# B&R Automation Studio project mVTest1
Automation Studio 4.12.6.106; technology packages: mappCockpit 5.24.2, mappMotion 5.29.0, mappView 5.24.6

## Configuration Config1

CPU X20CP3687X, AutomationRuntime J4.93, Build 4.1.2, Safety 0.0, Vc V4.73.2

### Task classes (Cpu.sw)
```
Cyclic#1:
  motionprg1 <- motionprg1.prg
  motionprg2 <- motionprg2.prg
Cyclic#4:
  Program <- Program.prg
DataObjects: McAcpSys
NcDataObjects: McDriveLog
Binaries: arsvcreg, udbdef, mvLoader, arflatprv, McAcpDrv, arcoal, FWRules, TCData, mCoWebSc, McAcpSim, Settings, Config_1, ashwac, User, sysconf, asfw, arconfig, Config_3, ashwd, Config_2, iomap, Role
Libraries: arssl, astime, asieccon, mpaxis, powerlnk, runtime, mcaxis, fileio, mpbase, mcbase, sys_lib, CoTrace, AsZip
```

### Hardware
```
X20CP3687X : X20CP3687X v1.6.2.0
  Connector IF2:
    ActivateDevice = 1
    Mode = Manual
    InternetAddress = 192.168.1.50
    SubnetMask = 255.255.255.0
  ConfigurationID = mVTest1_Config1
  FileDevice1
  FileDeviceName1 = USER
  FileDevicePath1 = USER_PATH
  ActivateOpcUa = 1
  OpcUa_AuthenticationSecurityPolicy_EnableNone = 1
  OpcUa_AuthenticationSecurityPolicy_EnableBasic128Rsa15 = 1
  OpcUaInformationModels_PV_Version = 1
```

### Config_2.axis - X20CP3687X/mappMotion/Config_2.axis
```
Element gAxis_2 (Type=axis)
  BaseTypeIsReadOnly = 0
  BaseType = Rotary
    MeasurementUnitIsReadOnly = 0
    MeasurementUnit = 17476
    MeasurementResolutionIsReadOnly = 0
    MeasurementResolution = 0.01
    CountDirectionIsReadOnly = 0
    CountDirection = Standard
  MovementLimitsIsReadOnly = 0
  MovementLimits = Internal
    Position:
      LowerLimitMin = -1.79769313486231E308
      UpperLimitMax = 1.79769313486231E308
      LowerLimit = -1000.0
      UpperLimit = 1000.0
    VelocityIsReadOnly = 0
    Velocity:
      VelocityMax = 3.4E38
      Velocity = 30
    AccelerationIsReadOnly = 0
    Acceleration:
      AccelerationMax = 3.4E38
      Acceleration = 50.0
    DecelerationIsReadOnly = 0
    Deceleration:
      DecelerationMax = 3.4E38
      Deceleration = 50.0
  Alarms = None
```

## Configuration Config2

CPU PC_any, AutomationRuntime J4.93, Build 4.1.2, Vc V4.73.2

### Hardware
```
PC : PC_any v1.1.1.0 (OrderNumber=PC)
  ConfigurationID = mVTest1_Config2
  FileDevice1
  FileDeviceName1 = USER
  FileDevicePath1 = USER_PATH
  ActivateOpcUa = 1
  OpcUaInformationModels_PV_Version = 1
```

## Configuration Config3

CPU 4PPC50.101E-10B, AutomationRuntime J4.93, Build 4.1.2, Safety 0.0, Vc V4.73.2

### Task classes (Cpu.sw)
```
Cyclic#1 (cycle 2000 us, tolerance 2000 us):
  motionprg1 <- motionprg1.prg
  motionprg2 <- motionprg2.prg
Cyclic#2 (cycle 20000 us, tolerance 20000 us):
  room3 <- room.prg
  room1 <- room.prg
  room2 <- room.prg
Cyclic#4 (cycle 100000 us, tolerance 100000 us):
  Program <- Program.prg
  tcp <- tcp.prg
DataObjects: McAcpSys
NcDataObjects: McDriveLog
Binaries: arsvcreg, udbdef, mvLoader, arflatprv, McAcpDrv, arcoal, FWRules, TCData, mCoWebSc, McAcpSim, Settings, Config_1, ashwac, User, sysconf, asfw, arconfig, iomap, Config_3, ashwd, Config_2, Role
Libraries: McBase, MpBase, MpAxis, McAxis, McAcpAx, CoTrace, AsZip, FileIO, runtime, AsTCP, helper, arssl, astime, asieccon, powerlnk, asepl, sys_lib
```

### Hardware
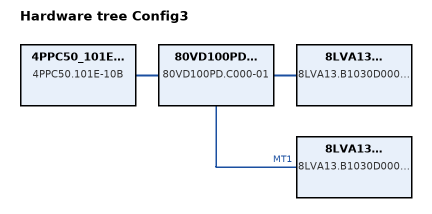
```
4PPC50_101E_10B : 4PPC50.101E-10B v1.1.4.0
  Connector IF2:
    ActivateDevice = 1
    Mode = Manual
    InternetAddress = 192.168.1.50
    SubnetMask = 255.255.255.0
    ActivateSnmp = 1
  Connector IF3:
    AssignedOperatingSystem = ARemb
  Connector IF4:
    AssignedOperatingSystem = GPOS
  ConfigurationID = mVTest1_Config3
  TimerDeviceType = EPLX2X
  TimerDevice = 4PPC50_101E_10B.IF1
  TaskClassIdleTime = 2000
  Cyclic1Duration = 2000
  Cyclic1Tolerance = 2000
  Cyclic2Duration = 20000
  Cyclic2Tolerance = 20000
  Cyclic3Duration = 50000
  Cyclic3Tolerance = 50000
  Cyclic4Duration = 100000
  Cyclic4Tolerance = 100000
  Cyclic5Duration = 200000
  Cyclic5Tolerance = 200000
  Cyclic6Duration = 500000
  Cyclic6Tolerance = 500000
  Cyclic7Duration = 1000000
  Cyclic7Tolerance = 1000000
  Cyclic8Duration = 10000
  Cyclic8Tolerance = 30000000
  FileDevice1
  FileDeviceName1 = USER
  FileDevicePath1 = USER_PATH
  ActivateOpcUa = 1
  OpcUa_AuthenticationSecurityPolicy_EnableNone = 1
  OpcUa_AuthenticationSecurityPolicy_EnableBasic128Rsa15 = 1
  OpcUaInformationModels_PV_Version = 1
  LXTMode = Manual
  LXTInternetAddress = 192.168.1.51
  LXTSubnetmask = 255.255.255.0
  LXTVisuURL = 192.168.1.50:81/index.html
80VD100PD.C000-01 : 80VD100PD.C000-01 v2.5.0.0  [PLK1 -> 4PPC50_101E_10B.IF1 (NodeNumber=1) [Cable Type=PowerlinkCable, Length=10, Version=1.0.0.3]; MT2 -> 8LVA13.B1030D000-0.MT]
  DriveConfiguration/Module:
    McAcoposTypeID = AcoposMicroDConfig
    ActivateACOPOSSimulationOnPLC = 0
  DriveConfiguration/Channel[1]/RealAxis:
    AxisReference = gAxis_1
    MechanicalElementsIsInvisible = 0
  DriveConfiguration/Channel[1]/RealAxis/MechanicalElements/Gearbox:
    InputIsReadOnly = 0
    Input = 1
    OutputIsReadOnly = 0
    Output = 1
  DriveConfiguration/Channel[1]/RealAxis/MechanicalElements/RotaryToLinearTransformation:
    ReferenceDistanceIsReadOnly = 0
    ReferenceDistance = 1
  DriveConfiguration/Channel[1]/RealAxis/Controller:
    ModeIsReadOnly = 0
    Mode = PositionController
  DriveConfiguration/Channel[1]/RealAxis/Controller/Mode/Position:
    ProportionalGain = 50.0
    IntegrationTime = 0.0
    PredictionTime = 0.0004
    TotalDelayTime = 0.0004
  DriveConfiguration/Channel[1]/RealAxis/Controller/Mode/Speed:
    ProportionalGainIsReadOnly = 0
    ProportionalGain = 2.0
    IntegrationTimeIsReadOnly = 0
    IntegrationTime = 0.0
    FilterTimeIsReadOnly = 0
    FilterTime = 0.0
  DriveConfiguration/Channel[1]/RealAxis/Controller/Mode/LoopFilters:
    LoopFilterXIsReadOnly = 0
    LoopFilter1 = NotUsed
    LoopFilter2 = NotUsed
    LoopFilter3 = NotUsed
  DriveConfiguration/Channel[1]/RealAxis/Homing:
    ModeIsReadOnly = 0
    Mode = Direct
  DriveConfiguration/Channel[1]/RealAxis/Homing/Mode:
    Position = 0.0
    ReferencePulse = NotUsed
  DriveConfiguration/Channel[1]/RealAxis/Homing:
    RestorePositionVariable = 
  DriveConfiguration/Channel[1]/RealAxis/StopReaction:
    QuickstopIsReadOnly = 0
    Quickstop = DecelerationLimit
    DriveErrorIsReadOnly = 0
    DriveError = DecelerationLimit
    FilterTime = 10
  DriveConfiguration/Channel[1]/RealAxis/MovementErrorLimits:
    PositionError = 10
    VelocityErrorMonitoring = Automatic1
  DriveConfiguration/Channel[1]/RealAxis:
    JerkFilterIsReadOnly = 0
    JerkFilter = NotUsed
    ZeroVibrationFilter = NotUsed
  DriveConfiguration/Channel[1]/RealAxis/DigitalInputs/HomingSwitch:
    SourceIsReadOnly = 0
    Source = NotUsed
    Level = High
  DriveConfiguration/Channel[1]/RealAxis/DigitalInputs/PositiveLimitSwitch:
    SourceIsReadOnly = 0
    Source = NotUsed
    Level = High
  DriveConfiguration/Channel[1]/RealAxis/DigitalInputs/NegativeLimitSwitch:
    SourceIsReadOnly = 0
    Source = NotUsed
    Level = High
  DriveConfiguration/Channel[1]/RealAxis/DigitalInputs/Trigger1:
    Source = Force
    Level = High
  DriveConfiguration/Channel[1]/RealAxis/DigitalInputs/Trigger2:
    Source = Force
    Level = High
  DriveConfiguration/Channel[1]/RealAxis/DigitalInputs/Quickstop:
    Input = NotUsed
  DriveConfiguration/Channel[1]/RealAxis/Simulation:
    SimulationModeOnPLC = SetValueGeneration
    SimulationModeOnACOPOS = NotUsed
  DriveConfiguration/Channel[1]:
    ExternalEncoderAxis = NotUsed
  DriveConfiguration/Channel[2]/RealAxis:
    AxisReference = gAxis_2
    MechanicalElementsIsInvisible = 0
  DriveConfiguration/Channel[2]/RealAxis/MechanicalElements/Gearbox:
    InputIsReadOnly = 0
    Input = 1
    OutputIsReadOnly = 0
    Output = 1
  DriveConfiguration/Channel[2]/RealAxis/MechanicalElements/RotaryToLinearTransformation:
    ReferenceDistanceIsReadOnly = 0
    ReferenceDistance = 1
  DriveConfiguration/Channel[2]/RealAxis/Controller:
    ModeIsReadOnly = 0
    Mode = PositionController
  DriveConfiguration/Channel[2]/RealAxis/Controller/Mode/Position:
    ProportionalGain = 50.0
    IntegrationTime = 0.0
    PredictionTime = 0.0004
    TotalDelayTime = 0.0004
  DriveConfiguration/Channel[2]/RealAxis/Controller/Mode/Speed:
    ProportionalGainIsReadOnly = 0
    ProportionalGain = 2.0
    IntegrationTimeIsReadOnly = 0
    IntegrationTime = 0.0
    FilterTimeIsReadOnly = 0
    FilterTime = 0.0
  DriveConfiguration/Channel[2]/RealAxis/Controller/Mode/LoopFilters:
    LoopFilterXIsReadOnly = 0
    LoopFilter1 = NotUsed
    LoopFilter2 = NotUsed
    LoopFilter3 = NotUsed
  DriveConfiguration/Channel[2]/RealAxis/Homing:
    ModeIsReadOnly = 0
    Mode = Direct
  DriveConfiguration/Channel[2]/RealAxis/Homing/Mode:
    Position = 0.0
    ReferencePulse = NotUsed
  DriveConfiguration/Channel[2]/RealAxis/Homing:
    RestorePositionVariable = 
  DriveConfiguration/Channel[2]/RealAxis/StopReaction:
    QuickstopIsReadOnly = 0
    Quickstop = DecelerationLimit
    DriveErrorIsReadOnly = 0
    DriveError = DecelerationLimit
    FilterTime = 0.0
  DriveConfiguration/Channel[2]/RealAxis/MovementErrorLimits:
    PositionError = 10
    VelocityErrorMonitoring = Automatic1
  DriveConfiguration/Channel[2]/RealAxis:
    JerkFilterIsReadOnly = 0
    JerkFilter = NotUsed
    ZeroVibrationFilter = NotUsed
  DriveConfiguration/Channel[2]/RealAxis/DigitalInputs/HomingSwitch:
    SourceIsReadOnly = 0
    Source = NotUsed
    Level = High
  DriveConfiguration/Channel[2]/RealAxis/DigitalInputs/PositiveLimitSwitch:
    SourceIsReadOnly = 0
    Source = NotUsed
    Level = High
  DriveConfiguration/Channel[2]/RealAxis/DigitalInputs/NegativeLimitSwitch:
    SourceIsReadOnly = 0
    Source = NotUsed
    Level = High
  DriveConfiguration/Channel[2]/RealAxis/DigitalInputs/Trigger1:
    Source = X2Trigger1
    Level = High
  DriveConfiguration/Channel[2]/RealAxis/DigitalInputs/Trigger2:
    Source = X2Trigger2
    Level = High
  DriveConfiguration/Channel[2]/RealAxis/DigitalInputs/Quickstop:
    Input = NotUsed
  DriveConfiguration/Channel[2]/RealAxis/Simulation:
    SimulationModeOnPLC = SetValueGeneration
    SimulationModeOnACOPOS = NotUsed
  DriveConfiguration/Channel[2]:
    ExternalEncoderAxis = NotUsed
8LVA13.B1030D000-0 : 8LVA13.B1030D000-0 v2.2.0.3  [MT -> 80VD100PD.C000-01.MT2]
  M1/MotorParameters:
    MOTOR_AMB_TEMP_RATED = 40
8LVA13.B1030D000-0a : 8LVA13.B1030D000-0 v2.2.0.3  [MT -> 80VD100PD.C000-01.MT1]
  M1/MotorParameters:
    MOTOR_AMB_TEMP_RATED = 40
```

### Config_1.axis - 4PPC50_101E_10B/mappMotion/Config_1.axis
```
Element gAxis_1 (Type=axis)
  BaseTypeIsReadOnly = 0
  BaseType = Rotary
    MeasurementUnitIsReadOnly = 0
    MeasurementUnit = 17476
    MeasurementResolutionIsReadOnly = 0
    MeasurementResolution = 0.01
    CountDirectionIsReadOnly = 0
    CountDirection = Standard
  MovementLimitsIsReadOnly = 0
  MovementLimits = Internal
    Position:
      LowerLimitMin = -1.79769313486231E308
      UpperLimitMax = 1.79769313486231E308
      LowerLimit = -1000.0
      UpperLimit = 1000.0
    VelocityIsReadOnly = 0
    Velocity:
      VelocityMax = 3.4E38
      Velocity = 10.0
    AccelerationIsReadOnly = 0
    Acceleration:
      AccelerationMax = 3.4E38
      Acceleration = 50.0
    DecelerationIsReadOnly = 0
    Deceleration:
      DecelerationMax = 3.4E38
      Deceleration = 50.0
  Alarms = None
```

### Config_2.axis - 4PPC50_101E_10B/mappMotion/Config_2.axis
```
Element gAxis_2 (Type=axis)
  BaseTypeIsReadOnly = 0
  BaseType = Rotary
    MeasurementUnitIsReadOnly = 0
    MeasurementUnit = 17476
    MeasurementResolutionIsReadOnly = 0
    MeasurementResolution = 0.01
    CountDirectionIsReadOnly = 0
    CountDirection = Standard
  MovementLimitsIsReadOnly = 0
  MovementLimits = Internal
    Position:
      LowerLimitMin = -1.79769313486231E308
      UpperLimitMax = 1.79769313486231E308
      LowerLimit = -1000.0
      UpperLimit = 1000.0
    VelocityIsReadOnly = 0
    Velocity:
      VelocityMax = 3.4E38
      Velocity = 10.0
    AccelerationIsReadOnly = 0
    Acceleration:
      AccelerationMax = 3.4E38
      Acceleration = 50.0
    DecelerationIsReadOnly = 0
    Deceleration:
      DecelerationMax = 3.4E38
      Deceleration = 50.0
  Alarms = None
```

## Configuration Config4

CPU 4PPC80.101E-11A, AutomationRuntime J4.93, Build 4.1.2, Safety 0.0, Vc V4.73.2

### Task classes (Cpu.sw)
```
Cyclic#1 (cycle 2000 us, tolerance 2000 us):
  motionprg1 <- motionprg1.prg
  motionprg2 <- motionprg2.prg
Cyclic#2:
  opctest <- opctest.prg
  room1 <- room.prg
  room3 <- room.prg
  room2 <- room.prg
Cyclic#4:
  Program <- Program.prg
  tcp <- tcp.prg
DataObjects: McAcpSys
NcDataObjects: McDriveLog
Binaries: arsvcreg, udbdef, mvLoader, arflatprv, McAcpDrv, arcoal, FWRules, TCData, mCoWebSc, McAcpSim, Settings, Config_1, ashwac, User, sysconf, asfw, arconfig, iomap, Config_3, ashwd, Config_2, Role
Libraries: McBase, MpBase, MpAxis, McAxis, McAcpAx, CoTrace, AsZip, FileIO, runtime, McAcpPar, sys_lib, brsystem, helper, arssl, astime, asieccon, powerlnk, asepl
```

### Hardware
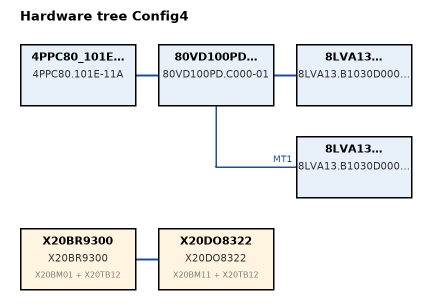
```
4PPC80_101E_11A : 4PPC80.101E-11A v1.0.3.0
  Connector IF2:
    AssignedOperatingSystem = ARemb
    ActivateDevice = 1
    Mode = Manual
    InternetAddress = 192.168.1.51
    SubnetMask = 255.255.255.0
    ActivateSnmp = 1
  Connector IF3:
    OperatingSystem = ARemb
    ActivateDevice = 1
  Connector IF4:
    AssignedOperatingSystem = GPOS
  Connector IF5:
    AssignedOperatingSystem = GPOS
  Connector IF6:
    CycleTime = 4000
  ConfigurationID = mVTest1_Config3
  TimerDeviceType = EPLX2X
  TimerDevice = 4PPC80_101E_11A.IF1
  TaskClassIdleTime = 2000
  Cyclic1Duration = 2000
  Cyclic1Tolerance = 2000
  FileDevice1
  FileDeviceName1 = USER
  FileDevicePath1 = USER_PATH
  ActivateOpcUa = 1
  OpcUa_AuthenticationSecurityPolicy_EnableNone = 1
  OpcUa_AuthenticationSecurityPolicy_EnableBasic128Rsa15 = 1
  OpcUaInformationModels_PV_Version = 1
  LXTVisuURL = 192.168.1.51:81/index.html
80VD100PD.C000-01 : 80VD100PD.C000-01 v2.5.0.0  [PLK1 -> 4PPC80_101E_11A.IF1 (NodeNumber=2) [Cable Type=PowerlinkCable, Length=10, Version=1.0.0.3]; MT2 -> 8LVA13.B1030D000-0.MT]
  DriveConfiguration/Module:
    McAcoposTypeID = AcoposMicroDConfig
    ActivateACOPOSSimulationOnPLC = 0
  DriveConfiguration/Channel[1]/RealAxis:
    AxisReference = gAxis_1
    MechanicalElementsIsInvisible = 0
  DriveConfiguration/Channel[1]/RealAxis/MechanicalElements/Gearbox:
    InputIsReadOnly = 0
    Input = 1
    OutputIsReadOnly = 0
    Output = 1
  DriveConfiguration/Channel[1]/RealAxis/MechanicalElements/RotaryToLinearTransformation:
    ReferenceDistanceIsReadOnly = 0
    ReferenceDistance = 1
  DriveConfiguration/Channel[1]/RealAxis/Controller:
    ModeIsReadOnly = 0
    Mode = PositionController
  DriveConfiguration/Channel[1]/RealAxis/Controller/Mode/Position:
    ProportionalGain = 50.0
    IntegrationTime = 0.0
    PredictionTime = 0.0004
    TotalDelayTime = 0.0004
  DriveConfiguration/Channel[1]/RealAxis/Controller/Mode/Speed:
    ProportionalGainIsReadOnly = 0
    ProportionalGain = 2.0
    IntegrationTimeIsReadOnly = 0
    IntegrationTime = 0.0
    FilterTimeIsReadOnly = 0
    FilterTime = 0.0
  DriveConfiguration/Channel[1]/RealAxis/Controller/Mode/LoopFilters:
    LoopFilterXIsReadOnly = 0
    LoopFilter1 = NotUsed
    LoopFilter2 = NotUsed
    LoopFilter3 = NotUsed
  DriveConfiguration/Channel[1]/RealAxis/Homing:
    ModeIsReadOnly = 0
    Mode = Direct
  DriveConfiguration/Channel[1]/RealAxis/Homing/Mode:
    Position = 0.0
    ReferencePulse = NotUsed
  DriveConfiguration/Channel[1]/RealAxis/Homing:
    RestorePositionVariable = 
  DriveConfiguration/Channel[1]/RealAxis/StopReaction:
    QuickstopIsReadOnly = 0
    Quickstop = DecelerationLimit
    DriveErrorIsReadOnly = 0
    DriveError = DecelerationLimit
    FilterTime = 10
  DriveConfiguration/Channel[1]/RealAxis/MovementErrorLimits:
    PositionError = 10
    VelocityErrorMonitoring = Automatic1
  DriveConfiguration/Channel[1]/RealAxis:
    JerkFilterIsReadOnly = 0
    JerkFilter = NotUsed
    ZeroVibrationFilter = NotUsed
  DriveConfiguration/Channel[1]/RealAxis/DigitalInputs/HomingSwitch:
    SourceIsReadOnly = 0
    Source = NotUsed
    Level = High
  DriveConfiguration/Channel[1]/RealAxis/DigitalInputs/PositiveLimitSwitch:
    SourceIsReadOnly = 0
    Source = NotUsed
    Level = High
  DriveConfiguration/Channel[1]/RealAxis/DigitalInputs/NegativeLimitSwitch:
    SourceIsReadOnly = 0
    Source = NotUsed
    Level = High
  DriveConfiguration/Channel[1]/RealAxis/DigitalInputs/Trigger1:
    Source = Force
    Level = High
  DriveConfiguration/Channel[1]/RealAxis/DigitalInputs/Trigger2:
    Source = Force
    Level = High
  DriveConfiguration/Channel[1]/RealAxis/DigitalInputs/Quickstop:
    Input = NotUsed
  DriveConfiguration/Channel[1]/RealAxis/Simulation:
    SimulationModeOnPLC = SetValueGeneration
    SimulationModeOnACOPOS = NotUsed
  DriveConfiguration/Channel[1]:
    ExternalEncoderAxis = NotUsed
  DriveConfiguration/Channel[2]/RealAxis:
    AxisReference = gAxis_2
    MechanicalElementsIsInvisible = 0
  DriveConfiguration/Channel[2]/RealAxis/MechanicalElements/Gearbox:
    InputIsReadOnly = 0
    Input = 1
    OutputIsReadOnly = 0
    Output = 1
  DriveConfiguration/Channel[2]/RealAxis/MechanicalElements/RotaryToLinearTransformation:
    ReferenceDistanceIsReadOnly = 0
    ReferenceDistance = 1
  DriveConfiguration/Channel[2]/RealAxis/Controller:
    ModeIsReadOnly = 0
    Mode = PositionController
  DriveConfiguration/Channel[2]/RealAxis/Controller/Mode/Position:
    ProportionalGain = 50.0
    IntegrationTime = 0.0
    PredictionTime = 0.0004
    TotalDelayTime = 0.0004
  DriveConfiguration/Channel[2]/RealAxis/Controller/Mode/Speed:
    ProportionalGainIsReadOnly = 0
    ProportionalGain = 2.0
    IntegrationTimeIsReadOnly = 0
    IntegrationTime = 0.0
    FilterTimeIsReadOnly = 0
    FilterTime = 0.0
  DriveConfiguration/Channel[2]/RealAxis/Controller/Mode/LoopFilters:
    LoopFilterXIsReadOnly = 0
    LoopFilter1 = NotUsed
    LoopFilter2 = NotUsed
    LoopFilter3 = NotUsed
  DriveConfiguration/Channel[2]/RealAxis/Homing:
    ModeIsReadOnly = 0
    Mode = Direct
  DriveConfiguration/Channel[2]/RealAxis/Homing/Mode:
    Position = 0.0
    ReferencePulse = NotUsed
  DriveConfiguration/Channel[2]/RealAxis/Homing:
    RestorePositionVariable = 
  DriveConfiguration/Channel[2]/RealAxis/StopReaction:
    QuickstopIsReadOnly = 0
    Quickstop = DecelerationLimit
    DriveErrorIsReadOnly = 0
    DriveError = DecelerationLimit
    FilterTime = 0.0
  DriveConfiguration/Channel[2]/RealAxis/MovementErrorLimits:
    PositionError = 10
    VelocityErrorMonitoring = Automatic1
  DriveConfiguration/Channel[2]/RealAxis:
    JerkFilterIsReadOnly = 0
    JerkFilter = NotUsed
    ZeroVibrationFilter = NotUsed
  DriveConfiguration/Channel[2]/RealAxis/DigitalInputs/HomingSwitch:
    SourceIsReadOnly = 0
    Source = NotUsed
    Level = High
  DriveConfiguration/Channel[2]/RealAxis/DigitalInputs/PositiveLimitSwitch:
    SourceIsReadOnly = 0
    Source = NotUsed
    Level = High
  DriveConfiguration/Channel[2]/RealAxis/DigitalInputs/NegativeLimitSwitch:
    SourceIsReadOnly = 0
    Source = NotUsed
    Level = High
  DriveConfiguration/Channel[2]/RealAxis/DigitalInputs/Trigger1:
    Source = X2Trigger1
    Level = High
  DriveConfiguration/Channel[2]/RealAxis/DigitalInputs/Trigger2:
    Source = X2Trigger2
    Level = High
  DriveConfiguration/Channel[2]/RealAxis/DigitalInputs/Quickstop:
    Input = NotUsed
  DriveConfiguration/Channel[2]/RealAxis/Simulation:
    SimulationModeOnPLC = SetValueGeneration
    SimulationModeOnACOPOS = NotUsed
  DriveConfiguration/Channel[2]:
    ExternalEncoderAxis = NotUsed
8LVA13.B1030D000-0 : 8LVA13.B1030D000-0 v2.2.0.3  [MT -> 80VD100PD.C000-01.MT2]
  M1/MotorParameters:
    MOTOR_AMB_TEMP_RATED = 40
8LVA13.B1030D000-0a : 8LVA13.B1030D000-0 v2.2.0.3  [MT -> 80VD100PD.C000-01.MT1]
  M1/MotorParameters:
    MOTOR_AMB_TEMP_RATED = 40
X20BM01 : X20BM01 v2.2.0.0
X20BM11 : X20BM11 v1.1.0.0  [X2X1 -> X20BM01.X2X2]
X20BR9300 : X20BR9300 v1.3.0.0  [SS1 -> X20TB12.SS; SL -> X20BM01.SL1; X2X1 -> 4PPC80_101E_11A.IF6 [Cable Type=X2XCable, Length=10, Version=1.0.0.3]]
X20DO8322 : X20DO8322 v1.5.0.0  [SS1 -> X20TB12a.SS; SL -> X20BM11.SL1]
X20TB12 : X20TB12 v1.0.0.0
X20TB12a : X20TB12 v1.0.0.0
```

## Configuration T50_X20CP0484

CPU X20CP0484, AutomationRuntime J4.93, Build 4.1.2, Safety 0.0, Vc 

### Task classes (Cpu.sw)
```
Cyclic#1 (cycle 2000 us, tolerance 0 us):
  motionprg1 <- motionprg1.prg
  motionprg2 <- motionprg2.prg
Cyclic#2 (cycle 20000 us, tolerance 20000 us):
  opctest <- opctest.prg
  room1 <- room.prg
  room2 <- room.prg
  room3 <- room.prg
  tcp <- tcp.prg
Cyclic#4 (cycle 100000 us, tolerance 100000 us):
  Program <- Program.prg
DataObjects: McAcpSys
NcDataObjects: McDriveLog
Binaries: FWRules, udbdef, TCData, arsvcreg, mvLoader, McAcpDrv, arflatprv, arcoal, mCoWebSc, McAcpSim, arconfig, asfw, iomap, Role, ashwd, ashwac, sysconf, User, Config_1, Config_3, Config_2, Settings, asnxdb2, asnxdb1
Libraries: Runtime, sys_lib, brsystem, FileIO, operator, AsTime, CoTrace, AsZip, helper, powerlnk, arssl, asieccon, mpaxis, mcaxis, mpbase, mcbase, asepl, mcacpax, astcp, asbrstr, asarcfg, vcresman, ashw
```

### Hardware
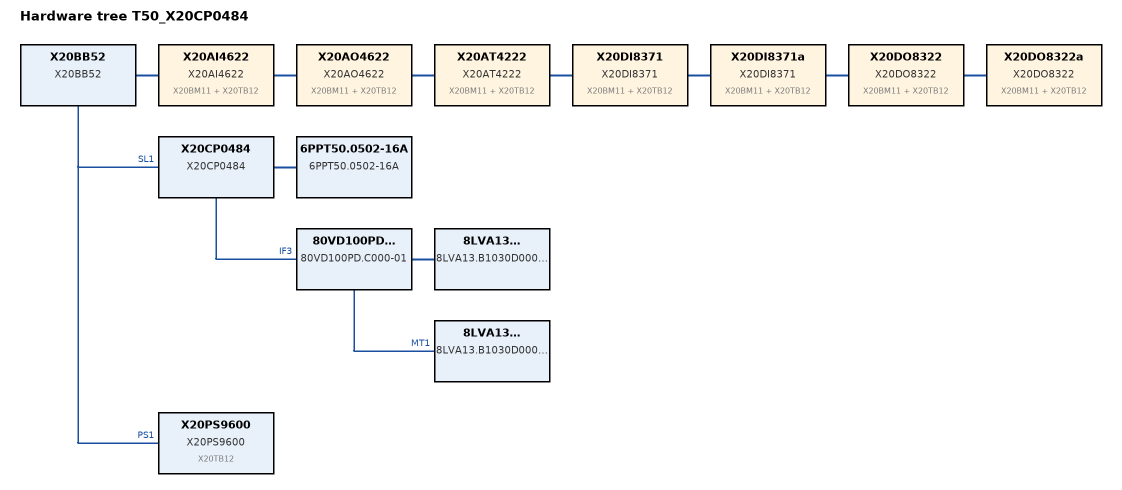
```
6PPT50.0502-16A : 6PPT50.0502-16A v1.3.8.0  [ETH2 -> X20CP0484.IF2 [Cable Type=PowerlinkCable, Length=10, Version=1.0.0.3]]
  Terminal = true
  PasswordVNC = 
  PasswordCIFS = 
  PasswordService = 
  VncVcObjectName = VisuW
  VncAuthentication = 1
  VncPasswordViewOnly = v
  VncPasswordViewControl = c
80VD100PD.C000-01 : 80VD100PD.C000-01 v2.5.0.0  [PLK1 -> X20CP0484.IF3 (NodeNumber=1) [Cable Type=PowerlinkCable, Length=10, Version=1.0.0.3]; MT2 -> 8LVA13.B1030D000-0.MT]
  DriveConfiguration/Module:
    McAcoposTypeID = AcoposMicroDConfig
    ActivateACOPOSSimulationOnPLC = 0
  DriveConfiguration/Channel[1]/RealAxis:
    AxisReference = gAxis_1
    MechanicalElementsIsInvisible = 0
  DriveConfiguration/Channel[1]/RealAxis/MechanicalElements/Gearbox:
    InputIsReadOnly = 0
    Input = 1
    OutputIsReadOnly = 0
    Output = 1
  DriveConfiguration/Channel[1]/RealAxis/MechanicalElements/RotaryToLinearTransformation:
    ReferenceDistanceIsReadOnly = 0
    ReferenceDistance = 1
  DriveConfiguration/Channel[1]/RealAxis/Controller:
    ModeIsReadOnly = 0
    Mode = PositionController
  DriveConfiguration/Channel[1]/RealAxis/Controller/Mode/Position:
    ProportionalGain = 50.0
    IntegrationTime = 0.0
    PredictionTime = 0.0004
    TotalDelayTime = 0.0004
  DriveConfiguration/Channel[1]/RealAxis/Controller/Mode/Speed:
    ProportionalGainIsReadOnly = 0
    ProportionalGain = 2.0
    IntegrationTimeIsReadOnly = 0
    IntegrationTime = 0.0
    FilterTimeIsReadOnly = 0
    FilterTime = 0.0
  DriveConfiguration/Channel[1]/RealAxis/Controller/Mode/LoopFilters:
    LoopFilterXIsReadOnly = 0
    LoopFilter1 = NotUsed
    LoopFilter2 = NotUsed
    LoopFilter3 = NotUsed
  DriveConfiguration/Channel[1]/RealAxis/Homing:
    ModeIsReadOnly = 0
    Mode = Direct
  DriveConfiguration/Channel[1]/RealAxis/Homing/Mode:
    Position = 0.0
    ReferencePulse = NotUsed
  DriveConfiguration/Channel[1]/RealAxis/Homing:
    RestorePositionVariable = 
  DriveConfiguration/Channel[1]/RealAxis/StopReaction:
    QuickstopIsReadOnly = 0
    Quickstop = DecelerationLimit
    DriveErrorIsReadOnly = 0
    DriveError = DecelerationLimit
    FilterTime = 10
  DriveConfiguration/Channel[1]/RealAxis/MovementErrorLimits:
    PositionError = 10
    VelocityErrorMonitoring = Automatic1
  DriveConfiguration/Channel[1]/RealAxis:
    JerkFilterIsReadOnly = 0
    JerkFilter = NotUsed
    ZeroVibrationFilter = NotUsed
  DriveConfiguration/Channel[1]/RealAxis/DigitalInputs/HomingSwitch:
    SourceIsReadOnly = 0
    Source = NotUsed
    Level = High
  DriveConfiguration/Channel[1]/RealAxis/DigitalInputs/PositiveLimitSwitch:
    SourceIsReadOnly = 0
    Source = NotUsed
    Level = High
  DriveConfiguration/Channel[1]/RealAxis/DigitalInputs/NegativeLimitSwitch:
    SourceIsReadOnly = 0
    Source = NotUsed
    Level = High
  DriveConfiguration/Channel[1]/RealAxis/DigitalInputs/Trigger1:
    Source = Force
    Level = High
  DriveConfiguration/Channel[1]/RealAxis/DigitalInputs/Trigger2:
    Source = Force
    Level = High
  DriveConfiguration/Channel[1]/RealAxis/DigitalInputs/Quickstop:
    Input = NotUsed
  DriveConfiguration/Channel[1]/RealAxis/Simulation:
    SimulationModeOnPLC = SetValueGeneration
    SimulationModeOnACOPOS = NotUsed
  DriveConfiguration/Channel[1]:
    ExternalEncoderAxis = NotUsed
  DriveConfiguration/Channel[2]/RealAxis:
    AxisReference = gAxis_2
    MechanicalElementsIsInvisible = 0
  DriveConfiguration/Channel[2]/RealAxis/MechanicalElements/Gearbox:
    InputIsReadOnly = 0
    Input = 1
    OutputIsReadOnly = 0
    Output = 1
  DriveConfiguration/Channel[2]/RealAxis/MechanicalElements/RotaryToLinearTransformation:
    ReferenceDistanceIsReadOnly = 0
    ReferenceDistance = 1
  DriveConfiguration/Channel[2]/RealAxis/Controller:
    ModeIsReadOnly = 0
    Mode = PositionController
  DriveConfiguration/Channel[2]/RealAxis/Controller/Mode/Position:
    ProportionalGain = 50.0
    IntegrationTime = 0.0
    PredictionTime = 0.0004
    TotalDelayTime = 0.0004
  DriveConfiguration/Channel[2]/RealAxis/Controller/Mode/Speed:
    ProportionalGainIsReadOnly = 0
    ProportionalGain = 2.0
    IntegrationTimeIsReadOnly = 0
    IntegrationTime = 0.0
    FilterTimeIsReadOnly = 0
    FilterTime = 0.0
  DriveConfiguration/Channel[2]/RealAxis/Controller/Mode/LoopFilters:
    LoopFilterXIsReadOnly = 0
    LoopFilter1 = NotUsed
    LoopFilter2 = NotUsed
    LoopFilter3 = NotUsed
  DriveConfiguration/Channel[2]/RealAxis/Homing:
    ModeIsReadOnly = 0
    Mode = Direct
  DriveConfiguration/Channel[2]/RealAxis/Homing/Mode:
    Position = 0.0
    ReferencePulse = NotUsed
  DriveConfiguration/Channel[2]/RealAxis/Homing:
    RestorePositionVariable = 
  DriveConfiguration/Channel[2]/RealAxis/StopReaction:
    QuickstopIsReadOnly = 0
    Quickstop = DecelerationLimit
    DriveErrorIsReadOnly = 0
    DriveError = DecelerationLimit
    FilterTime = 0.0
  DriveConfiguration/Channel[2]/RealAxis/MovementErrorLimits:
    PositionError = 10
    VelocityErrorMonitoring = Automatic1
  DriveConfiguration/Channel[2]/RealAxis:
    JerkFilterIsReadOnly = 0
    JerkFilter = NotUsed
    ZeroVibrationFilter = NotUsed
  DriveConfiguration/Channel[2]/RealAxis/DigitalInputs/HomingSwitch:
    SourceIsReadOnly = 0
    Source = NotUsed
    Level = High
  DriveConfiguration/Channel[2]/RealAxis/DigitalInputs/PositiveLimitSwitch:
    SourceIsReadOnly = 0
    Source = NotUsed
    Level = High
  DriveConfiguration/Channel[2]/RealAxis/DigitalInputs/NegativeLimitSwitch:
    SourceIsReadOnly = 0
    Source = NotUsed
    Level = High
  DriveConfiguration/Channel[2]/RealAxis/DigitalInputs/Trigger1:
    Source = X2Trigger1
    Level = High
  DriveConfiguration/Channel[2]/RealAxis/DigitalInputs/Trigger2:
    Source = X2Trigger2
    Level = High
  DriveConfiguration/Channel[2]/RealAxis/DigitalInputs/Quickstop:
    Input = NotUsed
  DriveConfiguration/Channel[2]/RealAxis/Simulation:
    SimulationModeOnPLC = SetValueGeneration
    SimulationModeOnACOPOS = NotUsed
  DriveConfiguration/Channel[2]:
    ExternalEncoderAxis = NotUsed
8LVA13.B1030D000-0 : 8LVA13.B1030D000-0 v2.2.0.3  [MT -> 80VD100PD.C000-01.MT2]
  M1/MotorParameters:
    MOTOR_AMB_TEMP_RATED = 40
8LVA13.B1030D000-0a : 8LVA13.B1030D000-0 v2.2.0.3  [MT -> 80VD100PD.C000-01.MT1]
  M1/MotorParameters:
    MOTOR_AMB_TEMP_RATED = 40
X20AI4622 : X20AI4622 v1.2.0.0  [SS1 -> X20TB12.SS; SL -> X20BM11.SL1]
X20AO4622 : X20AO4622 v1.3.0.0  [SS1 -> X20TB12a.SS; SL -> X20BM11a.SL1]
X20AT4222 : X20AT4222 v1.4.0.0  [SS1 -> X20TB12b.SS; SL -> X20BM11b.SL1]
X20BB52 : X20BB52 v1.2.0.0
  Connector IF6:
    CycleTime = 2000
X20BM11 : X20BM11 v1.1.0.0  [X2X1 -> X20BB52.IF6]
X20BM11a : X20BM11 v1.1.0.0  [X2X1 -> X20BM11.X2X2]
X20BM11b : X20BM11 v1.1.0.0  [X2X1 -> X20BM11a.X2X2]
X20BM11c : X20BM11 v1.1.0.0  [X2X1 -> X20BM11b.X2X2]
X20BM11d : X20BM11 v1.1.0.0  [X2X1 -> X20BM11c.X2X2]
X20BM11e : X20BM11 v1.1.0.0  [X2X1 -> X20BM11d.X2X2]
X20BM11f : X20BM11 v1.1.0.0  [X2X1 -> X20BM11e.X2X2]
X20CP0484 : X20CP0484 v1.6.0.0  [SL -> X20BB52.SL1]
  Connector IF2:
    ActivateDevice = 1
    HostName = unity_ds_ctrl
    Mode = Manual
    InternetAddress = 192.168.1.61
    SubnetMask = 255.255.255.0
  Connector IF3:
    DNAConfiguration = manual
  ConfigurationID = CoffeeMachine_T50_X20CP1586
  VolatileGlobalPvSize = 5000000
  TimerDeviceType = SWIOTIMER
  Cyclic1Duration = 2000
  Cyclic1Tolerance = 0
  Cyclic2Duration = 20000
  Cyclic2Tolerance = 20000
  Cyclic3Duration = 50000
  Cyclic3Tolerance = 50000
  Cyclic4Duration = 100000
  Cyclic4Tolerance = 100000
  Cyclic5Duration = 200000
  Cyclic5Tolerance = 200000
  Cyclic6Duration = 500000
  Cyclic6Tolerance = 500000
  Cyclic7Duration = 1000000
  Cyclic7Tolerance = 1000000
  Cyclic8Duration = 10000
  Cyclic8Tolerance = 30000000
  FileDevice1
  FileDeviceName1 = USER
  FileDevicePath1 = USER_PATH
  TimeZone = 140
  ActivateDaylightSavingTime = 1
  EthernetHostName = unity_ds_ctrl
  ActivateOpcUa = 1
  OpcUa_AuthenticationSecurityPolicy_EnableNone = 1
  OpcUa_AuthenticationSecurityPolicy_EnableBasic128Rsa15 = 1
  OpcUaInformationModels_PV_Version = 2
  OpcUaInformationModel_Facet = 0
  OpcUaInformationModel_TypeInformation = 0
  OpcUaInformationModel_BaseObjectTypeForStructures = 0
X20DI8371 : X20DI8371 v1.4.0.0  [SS1 -> X20TB12c.SS; SL -> X20BM11c.SL1]
X20DI8371a : X20DI8371 v1.4.0.0  [SS1 -> X20TB12d.SS; SL -> X20BM11d.SL1]
X20DO8322 : X20DO8322 v1.5.0.0  [SS1 -> X20TB12e.SS; SL -> X20BM11e.SL1]
X20DO8322a : X20DO8322 v1.5.0.0  [SS1 -> X20TB12f.SS; SL -> X20BM11f.SL1]
X20PS9600 : X20PS9600 v1.6.0.0  [PS -> X20BB52.PS1; SS1 -> X20TB12g.SS]
X20TB12 : X20TB12 v1.0.0.0
X20TB12a : X20TB12 v1.0.0.0
X20TB12b : X20TB12 v1.0.0.0
X20TB12c : X20TB12 v1.0.0.0
X20TB12d : X20TB12 v1.0.0.0
X20TB12e : X20TB12 v1.0.0.0
X20TB12f : X20TB12 v1.0.0.0
X20TB12g : X20TB12 v1.0.0.0
```

### IoMap.iom - X20CP0484/IoMap.iom
```iecst
VAR_CONFIG
	::room1:Lampe AT %QX."X20DO8322".DigitalOutput01;
	::room2:Lampe AT %QX."X20DO8322".DigitalOutput02;
	::room3:Lampe AT %QX."X20DO8322".DigitalOutput03;
	myDO04 AT %QX."X20DO8322".DigitalOutput04;
	myDO05 AT %QX."X20DO8322".DigitalOutput05;
	myDO06 AT %QX."X20DO8322".DigitalOutput06;
	myDO07 AT %QX."X20DO8322".DigitalOutput07;
	myDO08 AT %QX."X20DO8322".DigitalOutput08;
	myDO09 AT %QX."X20DO8322a".DigitalOutput01;
	myDO10 AT %QX."X20DO8322a".DigitalOutput02;
	myDO11 AT %QX."X20DO8322a".DigitalOutput03;
	myDO12 AT %QX."X20DO8322a".DigitalOutput04;
	myDO13 AT %QX."X20DO8322a".DigitalOutput05;
	myDO14 AT %QX."X20DO8322a".DigitalOutput06;
	myDO15 AT %QX."X20DO8322a".DigitalOutput07;
	myDO16 AT %QX."X20DO8322a".DigitalOutput08;
	::room1:SwitchValueHW AT %IX."X20DI8371".DigitalInput01;
	::room2:SwitchValueHW  AT %IX."X20DI8371".DigitalInput02;
	::room3:SwitchValueHW  AT %IX."X20DI8371".DigitalInput03;
END_VAR
```

## Configuration T50_X20CP1586mc

CPU X20CP1586, AutomationRuntime J4.93, Build 4.1.2, Safety 0.0, Vc 

### Task classes (Cpu.sw)
```
Cyclic#1 (cycle 2000 us, tolerance 0 us):
  motionprg1 <- motionprg1.prg
  motionprg2 <- motionprg2.prg
Cyclic#2:
  opctest <- opctest.prg
  room1 <- room.prg
  room2 <- room.prg
  room3 <- room.prg
Cyclic#4:
  Program <- Program.prg
  tcp <- tcp.prg
DataObjects: McAcpSys
NcDataObjects: McDriveLog
Binaries: FWRules, udbdef, TCData, arsvcreg, mvLoader, McAcpDrv, arflatprv, arcoal, mCoWebSc, McAcpSim, arconfig, asfw, iomap, Role, ashwd, ashwac, sysconf, User, Config_1, Config_3, Config_2, Settings, asnxdb2, asnxdb1
Libraries: Runtime, sys_lib, brsystem, FileIO, operator, AsTime, CoTrace, AsZip, powerlnk, arssl, asieccon, mpaxis, mcaxis, mpbase, mcbase, asepl, mcacpax, vcresman, ashw, helper
```

### Hardware
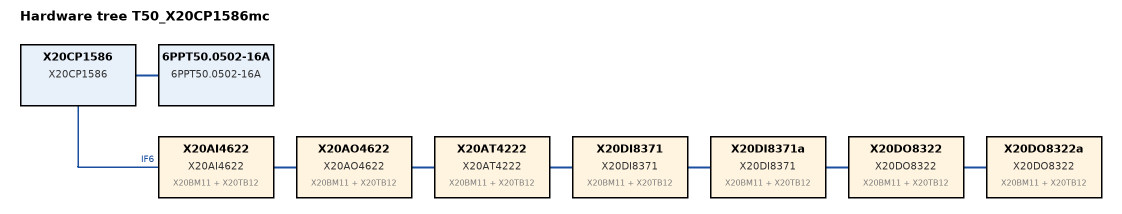
```
6PPT50.0502-16A : 6PPT50.0502-16A v1.3.8.0  [ETH2 -> X20CP1586.IF2 [Cable Type=PowerlinkCable, Length=10, Version=1.0.0.3]]
  Terminal = true
  PasswordVNC = 
  PasswordCIFS = 
  PasswordService = 
  VncVcObjectName = VisuW
  VncAuthentication = 1
  VncPasswordViewOnly = v
  VncPasswordViewControl = c
X20AI4622 : X20AI4622 v1.2.0.0  [SS1 -> X20TB12.SS; SL -> X20BM11.SL1]
X20AO4622 : X20AO4622 v1.3.0.0  [SS1 -> X20TB12a.SS; SL -> X20BM11a.SL1]
X20AT4222 : X20AT4222 v1.4.0.0  [SS1 -> X20TB12b.SS; SL -> X20BM11b.SL1]
X20BM11 : X20BM11 v1.1.0.0  [X2X1 -> X20CP1586.IF6]
X20BM11a : X20BM11 v1.1.0.0  [X2X1 -> X20BM11.X2X2]
X20BM11b : X20BM11 v1.1.0.0  [X2X1 -> X20BM11a.X2X2]
X20BM11c : X20BM11 v1.1.0.0  [X2X1 -> X20BM11b.X2X2]
X20BM11d : X20BM11 v1.1.0.0  [X2X1 -> X20BM11c.X2X2]
X20BM11e : X20BM11 v1.1.0.0  [X2X1 -> X20BM11d.X2X2]
X20BM11f : X20BM11 v1.1.0.0  [X2X1 -> X20BM11e.X2X2]
X20CP1586 : X20CP1586 v1.10.0.0
  Connector IF2:
    ActivateDevice = 1
    HostName = unity_ds_ctrl
    Mode = Manual
    InternetAddress = 192.168.1.61
    SubnetMask = 255.255.255.0
  Connector IF3:
    DNAConfiguration = manual
    EplHostName = unity_ds_ctrl
    HostName = unity_ds_ctrl
  ConfigurationID = CoffeeMachine_T50_X20CP1586
  VolatileGlobalPvSize = 5000000
  Cyclic1Duration = 2000
  Cyclic1Tolerance = 0
  FileDevice1
  FileDeviceName1 = USER
  FileDevicePath1 = USER_PATH
  TimeZone = 140
  ActivateDaylightSavingTime = 1
  EthernetHostName = unity_ds_ctrl
  ActivateOpcUa = 1
  OpcUa_AuthenticationSecurityPolicy_EnableNone = 1
  OpcUa_AuthenticationSecurityPolicy_EnableBasic128Rsa15 = 1
  OpcUaInformationModels_PV_Version = 2
  OpcUaInformationModel_Facet = 0
  OpcUaInformationModel_TypeInformation = 0
  OpcUaInformationModel_BaseObjectTypeForStructures = 0
X20DI8371 : X20DI8371 v1.4.0.0  [SS1 -> X20TB12c.SS; SL -> X20BM11c.SL1]
X20DI8371a : X20DI8371 v1.4.0.0  [SS1 -> X20TB12d.SS; SL -> X20BM11d.SL1]
X20DO8322 : X20DO8322 v1.5.0.0  [SS1 -> X20TB12e.SS; SL -> X20BM11e.SL1]
X20DO8322a : X20DO8322 v1.5.0.0  [SS1 -> X20TB12f.SS; SL -> X20BM11f.SL1]
X20TB12 : X20TB12 v1.0.0.0
X20TB12a : X20TB12 v1.0.0.0
X20TB12b : X20TB12 v1.0.0.0
X20TB12c : X20TB12 v1.0.0.0
X20TB12d : X20TB12 v1.0.0.0
X20TB12e : X20TB12 v1.0.0.0
X20TB12f : X20TB12 v1.0.0.0
```

## Configuration T50_X20CP3687Xmc

CPU X20CP3687X, AutomationRuntime J4.93, Build 4.1.2, Safety 0.0, Vc 

### Task classes (Cpu.sw)
```
Cyclic#1 (cycle 2000 us, tolerance 0 us):
  motionprg1 <- motionprg1.prg
  motionprg2 <- motionprg2.prg
Cyclic#2:
  opctest <- opctest.prg
  room1 <- room.prg
  room2 <- room.prg
  room3 <- room.prg
Cyclic#4:
  Program <- Program.prg
  tcp <- tcp.prg
DataObjects: McAcpSys
NcDataObjects: McDriveLog
Binaries: FWRules, udbdef, TCData, arsvcreg, mvLoader, McAcpDrv, arflatprv, arcoal, mCoWebSc, McAcpSim, arconfig, asfw, iomap, Role, ashwd, ashwac, sysconf, User, Config_1, Settings, Config_3, Config_2, asnxdb2, asnxdb1
Libraries: Runtime, sys_lib, brsystem, FileIO, operator, AsTime, CoTrace, AsZip, AsARCfg, AsMem, AsBrStr, helper, powerlnk, arssl, asieccon, mpaxis, mcaxis, mpbase, mcbase, asepl, mcacpax, vcresman, ashw
```

### Hardware
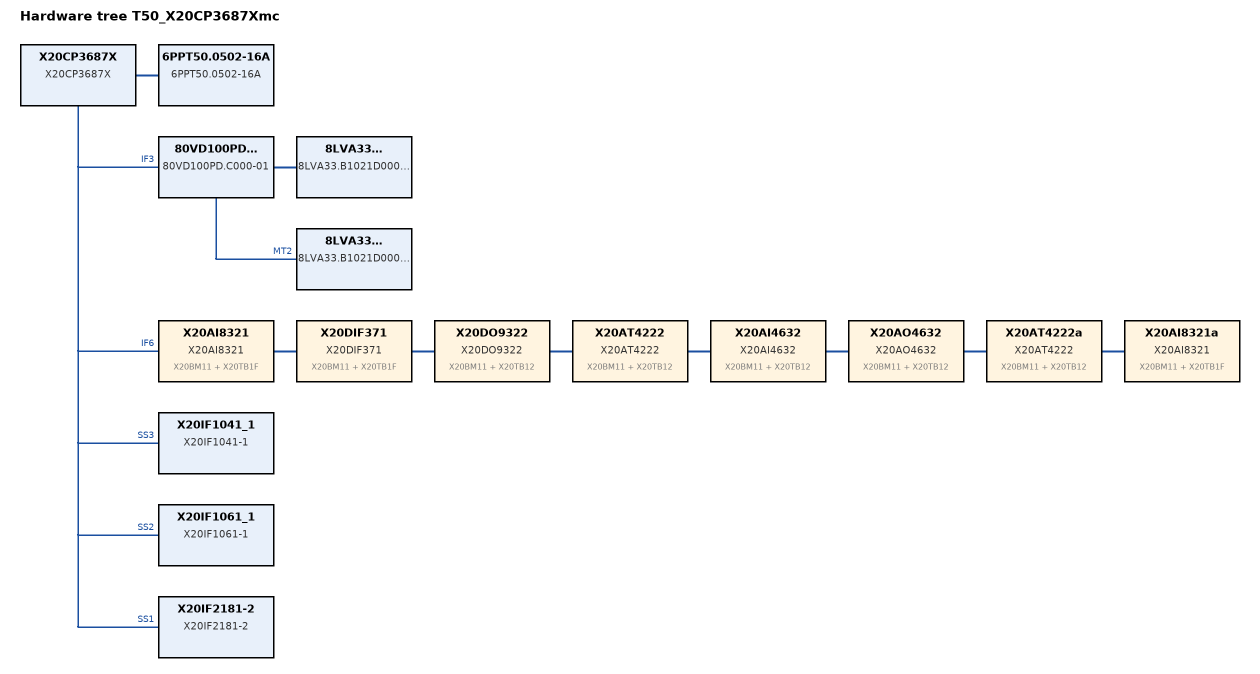
```
6PPT50.0502-16A : 6PPT50.0502-16A v1.3.8.0  [ETH2 -> X20CP3687X.IF2 [Cable Type=PowerlinkCable, Length=10, Version=1.0.0.3]]
  Terminal = true
  PasswordVNC = 
  PasswordCIFS = 
  PasswordService = 
  VncAuthentication = 1
  VncPasswordViewOnly = v
  VncPasswordViewControl = c
80VD100PD.C000-01 : 80VD100PD.C000-01 v2.5.0.0  [PLK1 -> X20CP3687X.IF3 (NodeNumber=1) [Cable Type=PowerlinkCable, Length=10, Version=1.0.0.3]; MT2 -> 8LVA33.B1021D000-0a.MT]
  DriveConfiguration/Module:
    McAcoposTypeID = AcoposMicroDConfig
    ActivateACOPOSSimulationOnPLC = 0
  DriveConfiguration/Channel[1]/RealAxis:
    AxisReference = gAxis_1
    MechanicalElementsIsInvisible = 0
  DriveConfiguration/Channel[1]/RealAxis/MechanicalElements/Gearbox:
    InputIsReadOnly = 0
    Input = 1
    OutputIsReadOnly = 0
    Output = 1
  DriveConfiguration/Channel[1]/RealAxis/MechanicalElements/RotaryToLinearTransformation:
    ReferenceDistanceIsReadOnly = 0
    ReferenceDistance = 1
  DriveConfiguration/Channel[1]/RealAxis/Controller:
    ModeIsReadOnly = 0
    Mode = PositionController
  DriveConfiguration/Channel[1]/RealAxis/Controller/Mode/Position:
    ProportionalGain = 50.0
    IntegrationTime = 0.0
    PredictionTime = 0.0004
    TotalDelayTime = 0.0004
  DriveConfiguration/Channel[1]/RealAxis/Controller/Mode/Speed:
    ProportionalGainIsReadOnly = 0
    ProportionalGain = 2.0
    IntegrationTimeIsReadOnly = 0
    IntegrationTime = 0.0
    FilterTimeIsReadOnly = 0
    FilterTime = 0.0
  DriveConfiguration/Channel[1]/RealAxis/Controller/Mode/LoopFilters:
    LoopFilterXIsReadOnly = 0
    LoopFilter1 = NotUsed
    LoopFilter2 = NotUsed
    LoopFilter3 = NotUsed
  DriveConfiguration/Channel[1]/RealAxis/Homing:
    ModeIsReadOnly = 0
    Mode = Direct
  DriveConfiguration/Channel[1]/RealAxis/Homing/Mode:
    Position = 0.0
    ReferencePulse = NotUsed
  DriveConfiguration/Channel[1]/RealAxis/Homing:
    RestorePositionVariable = 
  DriveConfiguration/Channel[1]/RealAxis/StopReaction:
    QuickstopIsReadOnly = 0
    Quickstop = DecelerationLimit
    DriveErrorIsReadOnly = 0
    DriveError = DecelerationLimit
    FilterTime = 10
  DriveConfiguration/Channel[1]/RealAxis/MovementErrorLimits:
    PositionError = 10
    VelocityErrorMonitoring = Automatic1
  DriveConfiguration/Channel[1]/RealAxis:
    JerkFilterIsReadOnly = 0
    JerkFilter = NotUsed
    ZeroVibrationFilter = NotUsed
  DriveConfiguration/Channel[1]/RealAxis/DigitalInputs/HomingSwitch:
    SourceIsReadOnly = 0
    Source = NotUsed
    Level = High
  DriveConfiguration/Channel[1]/RealAxis/DigitalInputs/PositiveLimitSwitch:
    SourceIsReadOnly = 0
    Source = NotUsed
    Level = High
  DriveConfiguration/Channel[1]/RealAxis/DigitalInputs/NegativeLimitSwitch:
    SourceIsReadOnly = 0
    Source = NotUsed
    Level = High
  DriveConfiguration/Channel[1]/RealAxis/DigitalInputs/Trigger1:
    Source = Force
    Level = High
  DriveConfiguration/Channel[1]/RealAxis/DigitalInputs/Trigger2:
    Source = Force
    Level = High
  DriveConfiguration/Channel[1]/RealAxis/DigitalInputs/Quickstop:
    Input = NotUsed
  DriveConfiguration/Channel[1]/RealAxis/Simulation:
    SimulationModeOnPLC = SetValueGeneration
    SimulationModeOnACOPOS = NotUsed
  DriveConfiguration/Channel[1]:
    ExternalEncoderAxis = NotUsed
  DriveConfiguration/Channel[2]/RealAxis:
    AxisReference = gAxis_2
    MechanicalElementsIsInvisible = 0
  DriveConfiguration/Channel[2]/RealAxis/MechanicalElements/Gearbox:
    InputIsReadOnly = 0
    Input = 1
    OutputIsReadOnly = 0
    Output = 1
  DriveConfiguration/Channel[2]/RealAxis/MechanicalElements/RotaryToLinearTransformation:
    ReferenceDistanceIsReadOnly = 0
    ReferenceDistance = 1
  DriveConfiguration/Channel[2]/RealAxis/Controller:
    ModeIsReadOnly = 0
    Mode = PositionController
  DriveConfiguration/Channel[2]/RealAxis/Controller/Mode/Position:
    ProportionalGain = 50.0
    IntegrationTime = 0.0
    PredictionTime = 0.0004
    TotalDelayTime = 0.0004
  DriveConfiguration/Channel[2]/RealAxis/Controller/Mode/Speed:
    ProportionalGainIsReadOnly = 0
    ProportionalGain = 2.0
    IntegrationTimeIsReadOnly = 0
    IntegrationTime = 0.0
    FilterTimeIsReadOnly = 0
    FilterTime = 0.0
  DriveConfiguration/Channel[2]/RealAxis/Controller/Mode/LoopFilters:
    LoopFilterXIsReadOnly = 0
    LoopFilter1 = NotUsed
    LoopFilter2 = NotUsed
    LoopFilter3 = NotUsed
  DriveConfiguration/Channel[2]/RealAxis/Homing:
    ModeIsReadOnly = 0
    Mode = Direct
  DriveConfiguration/Channel[2]/RealAxis/Homing/Mode:
    Position = 0.0
    ReferencePulse = NotUsed
  DriveConfiguration/Channel[2]/RealAxis/Homing:
    RestorePositionVariable = 
  DriveConfiguration/Channel[2]/RealAxis/StopReaction:
    QuickstopIsReadOnly = 0
    Quickstop = DecelerationLimit
    DriveErrorIsReadOnly = 0
    DriveError = DecelerationLimit
    FilterTime = 0.0
  DriveConfiguration/Channel[2]/RealAxis/MovementErrorLimits:
    PositionError = 10
    VelocityErrorMonitoring = Automatic1
  DriveConfiguration/Channel[2]/RealAxis:
    JerkFilterIsReadOnly = 0
    JerkFilter = NotUsed
    ZeroVibrationFilter = NotUsed
  DriveConfiguration/Channel[2]/RealAxis/DigitalInputs/HomingSwitch:
    SourceIsReadOnly = 0
    Source = NotUsed
    Level = High
  DriveConfiguration/Channel[2]/RealAxis/DigitalInputs/PositiveLimitSwitch:
    SourceIsReadOnly = 0
    Source = NotUsed
    Level = High
  DriveConfiguration/Channel[2]/RealAxis/DigitalInputs/NegativeLimitSwitch:
    SourceIsReadOnly = 0
    Source = NotUsed
    Level = High
  DriveConfiguration/Channel[2]/RealAxis/DigitalInputs/Trigger1:
    Source = X2Trigger1
    Level = High
  DriveConfiguration/Channel[2]/RealAxis/DigitalInputs/Trigger2:
    Source = X2Trigger2
    Level = High
  DriveConfiguration/Channel[2]/RealAxis/DigitalInputs/Quickstop:
    Input = NotUsed
  DriveConfiguration/Channel[2]/RealAxis/Simulation:
    SimulationModeOnPLC = SetValueGeneration
    SimulationModeOnACOPOS = NotUsed
  DriveConfiguration/Channel[2]:
    ExternalEncoderAxis = NotUsed
8LVA33.B1021D000-0 : 8LVA33.B1021D000-0 v2.2.0.3  [MT -> 80VD100PD.C000-01.MT1]
  M1/MotorParameters:
    MOTOR_AMB_TEMP_RATED = 40
8LVA33.B1021D000-0a : 8LVA33.B1021D000-0 v2.2.0.3  [MT -> 80VD100PD.C000-01.MT2]
  M1/MotorParameters:
    MOTOR_AMB_TEMP_RATED = 40
X20AI4632 : X20AI4632 v1.3.0.0  [SS1 -> X20TB12b.SS; SL -> X20BM11d.SL1]
  Supervision = off
X20AI8321 : X20AI8321 v1.5.0.0  [SS1 -> X20TB1F.SS; SL -> X20BM11.SL1]
  Supervision = off
X20AI8321a : X20AI8321 v1.5.0.0 (Disabled=true)  [SS1 -> X20TB1F2.SS; SL -> X20BM11g.SL1]
X20AO4632 : X20AO4632 v1.2.0.0  [SS1 -> X20TB12c.SS; SL -> X20BM11e.SL1]
  Supervision = off
X20AT4222 : X20AT4222 v1.4.0.0  [SS1 -> X20TB12a.SS; SL -> X20BM11c.SL1]
  Supervision = off
X20AT4222a : X20AT4222 v1.4.0.0 (Disabled=true)  [SS1 -> X20TB12d.SS; SL -> X20BM11f.SL1]
  Supervision = off
X20BM11 : X20BM11 v1.1.0.0  [X2X1 -> X20CP3687X.IF6]
X20BM11a : X20BM11 v1.1.0.0  [X2X1 -> X20BM11.X2X2]
X20BM11b : X20BM11 v1.1.0.0  [X2X1 -> X20BM11a.X2X2]
X20BM11c : X20BM11 v1.1.0.0  [X2X1 -> X20BM11b.X2X2]
X20BM11d : X20BM11 v1.1.0.0  [X2X1 -> X20BM11c.X2X2]
X20BM11e : X20BM11 v1.1.0.0  [X2X1 -> X20BM11d.X2X2]
X20BM11f : X20BM11 v1.1.0.0 (Disabled=true)  [X2X1 -> X20BM11e.X2X2]
X20BM11g : X20BM11 v1.1.0.0 (Disabled=true)  [X2X1 -> X20BM11f.X2X2]
X20CP3687X : X20CP3687X v1.6.2.0
  Connector IF2:
    ActivateDevice = 1
    HostName = unity_ds_ctrl
    Mode = Manual
    InternetAddress = 192.168.1.60
    SubnetMask = 255.255.255.0
    ActivateSnmp = 1
  Connector IF3:
    DNAConfiguration = manual
    EplHostName = unity_ds_ctrl
    CycleTime = 2000
    HostName = unity_ds_ctrl
  ConfigurationID = CoffeeMachine_T50_X20CP1586
  Cyclic1Duration = 2000
  Cyclic1Tolerance = 0
  FileDevice1
  FileDeviceName1 = USER
  FileDevicePath1 = USER_PATH
  TimeZone = 140
  ActivateDaylightSavingTime = 1
  EthernetHostName = unity_ds_ctrl
  ActivateOpcUa = 1
  OpcUa_AuthenticationSecurityPolicy_EnableNone = 1
  OpcUa_AuthenticationSecurityPolicy_EnableBasic128Rsa15 = 1
  OpcUaInformationModels_PV_Version = 2
  OpcUaInformationModel_Facet = 0
  OpcUaInformationModel_TypeInformation = 0
  OpcUaInformationModel_BaseObjectTypeForStructures = 0
X20DIF371 : X20DIF371 v1.3.0.0  [SS1 -> X20TB1F1.SS; SL -> X20BM11a.SL1]
  Supervision = off
X20DO9322 : X20DO9322 v1.5.0.0  [SS1 -> X20TB12.SS; SL -> X20BM11b.SL1]
  Supervision = off
X20IF1041_1 : X20IF1041-1 v1.4.0.0  [SS -> X20CP3687X.SS3]
  Connector IF1:
    DtmId = d18db546-0812-475b-a490-bf4d722b923f
  ConfigFile = X20IF1041_1.dtm
  ConfigModule = asnxdb2
  CycleTime = 2000
X20IF1061_1 : X20IF1061-1 v1.9.0.0  [SS -> X20CP3687X.SS2]
  Connector IF1:
    DtmId = c5118ea9-c0ff-4573-881d-1b306d6a3640
  ConfigFile = X20IF1061_1.dtm
  ConfigModule = asnxdb1
  CycleTime = 2000
X20IF2181-2 : X20IF2181-2 v1.9.0.0  [SS -> X20CP3687X.SS1]
  Connector IF1:
    EplNatSubnet = 192.168.102.0
X20TB12 : X20TB12 v1.0.0.0
X20TB12a : X20TB12 v1.0.0.0
X20TB12b : X20TB12 v1.0.0.0
X20TB12c : X20TB12 v1.0.0.0
X20TB12d : X20TB12 v1.0.0.0 (Disabled=true)
X20TB1F : X20TB1F v1.0.0.0
X20TB1F1 : X20TB1F v1.0.0.0
X20TB1F2 : X20TB1F v1.0.0.0 (Disabled=true)
```

### IoMap.iom - X20CP3687X/IoMap.iom
```iecst
VAR_CONFIG
	::room1:Lampe AT %QX."X20DO9322".DigitalOutput01;
	::room2:Lampe AT %QX."X20DO9322".DigitalOutput02;
	::room3:Lampe AT %QX."X20DO9322".DigitalOutput03;
	myDO04 AT %QX."X20DO9322".DigitalOutput04;
	myDO05 AT %QX."X20DO9322".DigitalOutput05;
	myDO06  AT %QX."X20DO9322".DigitalOutput06;
	myDO07  AT %QX."X20DO9322".DigitalOutput07;
	myDO08  AT %QX."X20DO9322".DigitalOutput08;
	myDO09  AT %QX."X20DO9322".DigitalOutput09;
	myDO10  AT %QX."X20DO9322".DigitalOutput10;
	myDO11  AT %QX."X20DO9322".DigitalOutput11;
	myDO12  AT %QX."X20DO9322".DigitalOutput12;
END_VAR
```

### Config_1.axis - X20CP3687X/mappMotion/Config_1.axis
```
Element gAxis_1 (Type=axis)
  BaseTypeIsReadOnly = 0
  BaseType = Rotary
    MeasurementUnitIsReadOnly = 0
    MeasurementUnit = 17476
    MeasurementResolutionIsReadOnly = 0
    MeasurementResolution = 0.01
    CountDirectionIsReadOnly = 0
    CountDirection = Standard
  MovementLimitsIsReadOnly = 0
  MovementLimits = Internal
    Position:
      LowerLimitMin = -1.79769313486231E308
      UpperLimitMax = 1.79769313486231E308
      LowerLimit = -1000.0
      UpperLimit = 1000.0
    VelocityIsReadOnly = 0
    Velocity:
      VelocityMax = 3.4E38
      Velocity = 30
    AccelerationIsReadOnly = 0
    Acceleration:
      AccelerationMax = 3.4E38
      Acceleration = 50.0
    DecelerationIsReadOnly = 0
    Deceleration:
      DecelerationMax = 3.4E38
      Deceleration = 50.0
  Alarms = None
```

## Configuration T50_X20CP3687XmcSim

CPU X20CP3687X, AutomationRuntime J4.93, Build 4.1.2, Safety 0.0, Vc 

### Task classes (Cpu.sw)
```
Cyclic#1 (cycle 2000 us, tolerance 0 us):
  motionprg1 <- motionprg1.prg
  motionprg2 <- motionprg2.prg
Cyclic#2:
  opctest <- opctest.prg
  room1 <- room.prg
  room2 <- room.prg
  room3 <- room.prg
Cyclic#4:
  Program <- Program.prg
  tcp <- tcp.prg
DataObjects: McAcpSys
NcDataObjects: McDriveLog
Binaries: FWRules, udbdef, TCData, arsvcreg, mvLoader, McAcpDrv, arflatprv, arcoal, mCoWebSc, McAcpSim, arconfig, asfw, iomap, Role, ashwd, ashwac, sysconf, User, Config_1, Settings, Config_3, Config_2, asnxdb2, asnxdb1
Libraries: Runtime, sys_lib, brsystem, FileIO, operator, AsTime, CoTrace, AsZip, powerlnk, arssl, asieccon, mpaxis, mcaxis, mpbase, mcbase, asepl, mcacpax, astcp, asbrstr, asarcfg, helper, vcresman, ashw
```

### Hardware
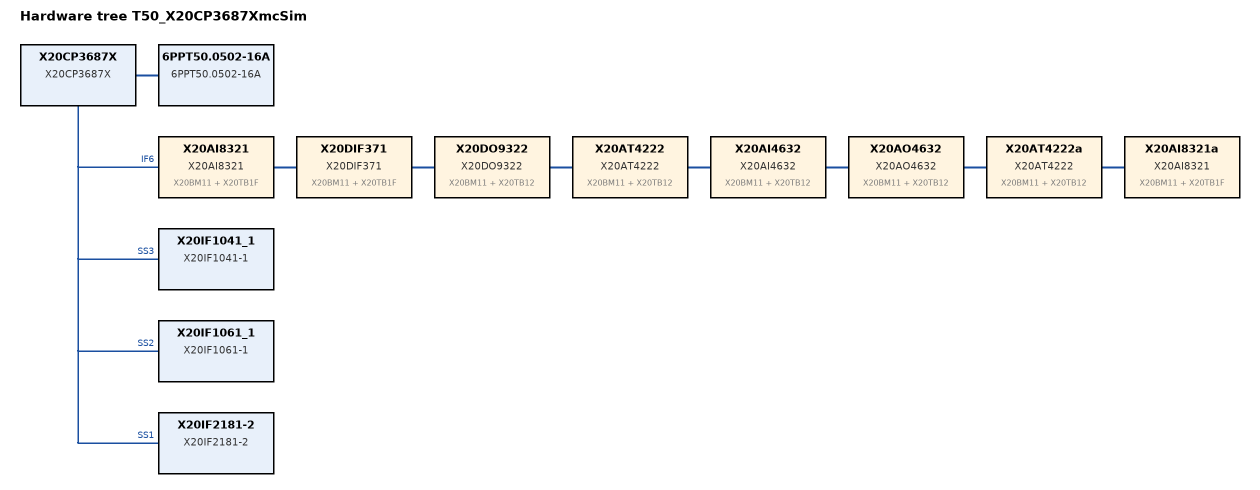
```
6PPT50.0502-16A : 6PPT50.0502-16A v1.3.8.0  [ETH2 -> X20CP3687X.IF2 [Cable Type=PowerlinkCable, Length=10, Version=1.0.0.3]]
  Terminal = true
  PasswordVNC = 
  PasswordCIFS = 
  PasswordService = 
  VncAuthentication = 1
  VncPasswordViewOnly = v
  VncPasswordViewControl = c
X20AI4632 : X20AI4632 v1.3.0.0  [SS1 -> X20TB12b.SS; SL -> X20BM11d.SL1]
  Supervision = off
X20AI8321 : X20AI8321 v1.5.0.0  [SS1 -> X20TB1F.SS; SL -> X20BM11.SL1]
  Supervision = off
X20AI8321a : X20AI8321 v1.5.0.0 (Disabled=true)  [SS1 -> X20TB1F2.SS; SL -> X20BM11g.SL1]
X20AO4632 : X20AO4632 v1.2.0.0  [SS1 -> X20TB12c.SS; SL -> X20BM11e.SL1]
  Supervision = off
X20AT4222 : X20AT4222 v1.4.0.0  [SS1 -> X20TB12a.SS; SL -> X20BM11c.SL1]
  Supervision = off
X20AT4222a : X20AT4222 v1.4.0.0 (Disabled=true)  [SS1 -> X20TB12d.SS; SL -> X20BM11f.SL1]
  Supervision = off
X20BM11 : X20BM11 v1.1.0.0  [X2X1 -> X20CP3687X.IF6]
X20BM11a : X20BM11 v1.1.0.0  [X2X1 -> X20BM11.X2X2]
X20BM11b : X20BM11 v1.1.0.0  [X2X1 -> X20BM11a.X2X2]
X20BM11c : X20BM11 v1.1.0.0  [X2X1 -> X20BM11b.X2X2]
X20BM11d : X20BM11 v1.1.0.0  [X2X1 -> X20BM11c.X2X2]
X20BM11e : X20BM11 v1.1.0.0  [X2X1 -> X20BM11d.X2X2]
X20BM11f : X20BM11 v1.1.0.0 (Disabled=true)  [X2X1 -> X20BM11e.X2X2]
X20BM11g : X20BM11 v1.1.0.0 (Disabled=true)  [X2X1 -> X20BM11f.X2X2]
X20CP3687X : X20CP3687X v1.6.2.0
  Connector IF2:
    ActivateDevice = 1
    HostName = unity_ds_ctrl
    Mode = Manual
    InternetAddress = 192.168.1.60
    SubnetMask = 255.255.255.0
    ActivateSnmp = 1
  Connector IF3:
    DNAConfiguration = manual
    EplHostName = unity_ds_ctrl
    CycleTime = 2000
    HostName = unity_ds_ctrl
  ConfigurationID = CoffeeMachine_T50_X20CP1586
  Simulation = 1
  Cyclic1Duration = 2000
  Cyclic1Tolerance = 0
  FileDevice1
  FileDeviceName1 = USER
  FileDevicePath1 = USER_PATH
  TimeZone = 140
  ActivateDaylightSavingTime = 1
  EthernetHostName = unity_ds_ctrl
  ActivateOpcUa = 1
  OpcUa_AuthenticationSecurityPolicy_EnableNone = 1
  OpcUa_AuthenticationSecurityPolicy_EnableBasic128Rsa15 = 1
  OpcUaInformationModels_PV_Version = 2
  OpcUaInformationModel_Facet = 0
  OpcUaInformationModel_TypeInformation = 0
  OpcUaInformationModel_BaseObjectTypeForStructures = 0
X20DIF371 : X20DIF371 v1.3.0.0  [SS1 -> X20TB1F1.SS; SL -> X20BM11a.SL1]
  Supervision = off
X20DO9322 : X20DO9322 v1.5.0.0  [SS1 -> X20TB12.SS; SL -> X20BM11b.SL1]
  Supervision = off
X20IF1041_1 : X20IF1041-1 v1.4.0.0  [SS -> X20CP3687X.SS3]
  Connector IF1:
    DtmId = d18db546-0812-475b-a490-bf4d722b923f
  ConfigFile = X20IF1041_1.dtm
  ConfigModule = asnxdb2
  CycleTime = 2000
X20IF1061_1 : X20IF1061-1 v1.9.0.0  [SS -> X20CP3687X.SS2]
  Connector IF1:
    DtmId = c5118ea9-c0ff-4573-881d-1b306d6a3640
  ConfigFile = X20IF1061_1.dtm
  ConfigModule = asnxdb1
  CycleTime = 2000
X20IF2181-2 : X20IF2181-2 v1.9.0.0  [SS -> X20CP3687X.SS1]
  Connector IF1:
    EplNatSubnet = 192.168.102.0
X20TB12 : X20TB12 v1.0.0.0
X20TB12a : X20TB12 v1.0.0.0
X20TB12b : X20TB12 v1.0.0.0
X20TB12c : X20TB12 v1.0.0.0
X20TB12d : X20TB12 v1.0.0.0 (Disabled=true)
X20TB1F : X20TB1F v1.0.0.0
X20TB1F1 : X20TB1F v1.0.0.0
X20TB1F2 : X20TB1F v1.0.0.0 (Disabled=true)
```

### IoMap.iom - X20CP3687X/IoMap.iom
```iecst
VAR_CONFIG
	::room1:Lampe AT %QX."X20DO9322".DigitalOutput01;
	::room2:Lampe AT %QX."X20DO9322".DigitalOutput02;
	::room3:Lampe AT %QX."X20DO9322".DigitalOutput03;
	myDO04 AT %QX."X20DO9322".DigitalOutput04;
	myDO05 AT %QX."X20DO9322".DigitalOutput05;
	myDO06 AT %QX."X20DO9322".DigitalOutput06;
	myDO07 AT %QX."X20DO9322".DigitalOutput07;
	myDO08 AT %QX."X20DO9322".DigitalOutput08;
	myDO09 AT %QX."X20DO9322".DigitalOutput09;
	myDO10 AT %QX."X20DO9322".DigitalOutput10;
	myDO11 AT %QX."X20DO9322".DigitalOutput11;
	myDO12 AT %QX."X20DO9322".DigitalOutput12;
END_VAR
```

### Config_3.axisfeature - X20CP3687X/mappMotion/Config_3.axisfeature
```
Element Feature_1 (Type=axisfeature)
  Type = CamAutomat
    CamAutomatType = ACOPOS
      CommonParameters:
        Master:
          ValueSource = SetPosition
            AxisReference
            MaxVelocity = 1.0
          StartPosition = 0.0
          StartInterval = MasterAxisPeriod
        AdvancedParameters:
          StartStateParameters:
            StartState = 0
            RelMasterStartPos = 0.0
          AdditiveAxes:
            AdditiveMasterValueSource = NotUsed
            AdditiveSlaveValueSource = NotUsed
          MasterStartPositionMode = NotEvaluatedAnew
          ControlSettings:
            CrossLeftBoundary = PositionLimitedHorizontal
            CamChangeImmediately = CurrentMasterMoveDir
          MessageSettings:
            ErrorsInStandby = NoErrorMessages
          TriggerAndLatch:
            Trigger1Delay = 0.0
            Trigger2Delay = 0.0
            SlaveLatchParID = 0
          EventParIDs
          StartIntervals
          Factors:
            SlaveFactorParID = 0
      States:
        State0 = Used
```

## Logical view

Binary libraries used (declarations not repeated): operator, runtime, astime, AsIecCon, McBase, MpBase, MpAxis, McAxis, McAcpAx, CoTrace, AsZip, FileIO, McAcpPar 5.29.0, sys_lib, brsystem, AsTCP, AsARCfg, AsMem, AsBrStr

### Global.var - Global variables
```iecst
VAR
	gVar1 : {REDUND_UNREPLICABLE} UDINT;
	gSetVar1 : {REDUND_UNREPLICABLE} BOOL;
	OPCUA_R1_Down : {REDUND_UNREPLICABLE} USINT;
	mV_R1_Down : {REDUND_UNREPLICABLE} USINT;
	OPCUA_R1_Up : {REDUND_UNREPLICABLE} USINT;
	mV_R1_Up : {REDUND_UNREPLICABLE} USINT;
	OPCUA_R2_Down : {REDUND_UNREPLICABLE} USINT;
	mV_R2_Down : {REDUND_UNREPLICABLE} USINT;
	OPCUA_R2_Up : {REDUND_UNREPLICABLE} USINT;
	mV_R2_Up : {REDUND_UNREPLICABLE} USINT;
END_VAR
VAR CONSTANT
	mcPOSITIVE_DIR : USINT := 0;
	mcNEGATIVE_DIR : USINT := 1;
END_VAR
VAR
	OPCUA_R1_Stop : USINT;
	mV_R1_Stop : USINT;
	gSchweibsWrite : REAL := 0.0;
	gSchweibsChange : REAL := 0.0;
	myDO01 : BOOL := 0;
	myDO02 : BOOL := 0;
	myDO03 : BOOL := 0;
	myDO04 : BOOL := 0;
	myDO06 : BOOL := 0;
	myDO05 : BOOL := 0;
	myDO07 : BOOL := 0;
	myDO08 : BOOL := 0;
	myDO09 : BOOL := 0;
	myDO10 : BOOL := 0;
	myDO11 : BOOL := 0;
	myDO12 : BOOL := 0;
	myDO13 : BOOL := 0;
	myDO14 : BOOL := 0;
	myDO15 : BOOL := 0;
	myDO16 : BOOL := 0;
	gDataSend : BOOL;
	gSendMessage : STRING[320];
	gGlassesOnline : {REDUND_UNREPLICABLE} BOOL;
	gTablettOnline : {REDUND_UNREPLICABLE} BOOL;
	gWindowsOnline : {REDUND_UNREPLICABLE} BOOL;
END_VAR
```

### Package Logical/Libraries - Global libraries

### Library Logical/Libraries/helper (ANSIC)

#### helper.fun - Exported functions and function blocks
```iecst
{REDUND_ERROR} FUNCTION findinstr : BOOL (*TODO: Add your comment here*) (*$GROUP=User,$CAT=User,$GROUPICON=User.png,$CATICON=User.png*)
	VAR_INPUT
		String1 : STRING[80];
		String2 : STRING[80];
	END_VAR
END_FUNCTION
```

#### findinstr.c
```c
#include <bur/plctypes.h>
#include <string.h>
#ifdef __cplusplus
	extern "C"
	{
#endif
	#include "helper.h"
#ifdef __cplusplus
	};
#endif
/* TODO: Add your comment here */
plcbit findinstr(plcstring* String1,plcstring* String2)
{
	/*TODO: Add your code here*/
	char * mysubstring = strstr(String1, String2);
	if (mysubstring != NULL) {
		return 1;
	}
	else
	{
		return 0;
	}
}
```

### Program Logical/Program (IEC)

#### Main.st
```iecst
PROGRAM _INIT
	(* Insert code here *)
	gSetVar1 := 0;
	gVar1 := 0;
END_PROGRAM

PROGRAM _CYCLIC
	(* Insert code here *)
	 gVar1 := gVar1 + 1;
END_PROGRAM

PROGRAM _EXIT
	(* Insert code here *)

END_PROGRAM
```

- Visualisation Logical/mappView (not shown)

### Program Logical/motionprg1 (IEC)

#### Variables.var
```iecst
VAR
	MpAxisBasic_0 : MpAxisBasic;
	AxisParameters : MpAxisBasicParType;
	McAcpAxProcessParIDType_var : {REDUND_UNREPLICABLE} McAcpAxProcessParIDType;
	ParId719Value : UDINT;
	MC_BR_ProcessParID_AcpAx_0 : MC_BR_ProcessParID_AcpAx;
	MC_BR_ProcessParID_AcpAx_Exe : BOOL;
	MC_MoveVelocity_0 : MC_MoveVelocity;
	MC_MoveVelocity_1 : MC_MoveVelocity;
	OPCUA_R1_Down_Cnt : UDINT;
END_VAR
```

#### Main.st
```iecst
PROGRAM _INIT

	MpAxisBasic_0.Enable := TRUE;
	MC_BR_ProcessParID_AcpAx_Exe := TRUE;

	AxisParameters.Position := 100.0;
	AxisParameters.Velocity := 10.0;
	AxisParameters.Acceleration := 50.0;
	AxisParameters.Deceleration := 50.0;

	ParId719Value := 1;
	McAcpAxProcessParIDType_var.DataType 		:= mcACPAX_PARTYPE_UDINT;
	McAcpAxProcessParIDType_var.ParID 			:= mcACPPAR_ENCOD_CMD;
	McAcpAxProcessParIDType_var.VariableAddress := ADR(ParId719Value);

END_PROGRAM

PROGRAM _CYCLIC

	MpAxisBasic_0.MpLink     					:= ADR(gAxis_1);
	MpAxisBasic_0.Parameters 					:= ADR(AxisParameters);
	MpAxisBasic_0();

	MC_BR_ProcessParID_AcpAx_0(Axis := ADR(gAxis_1), Execute := MC_BR_ProcessParID_AcpAx_Exe, DataAddress := ADR(McAcpAxProcessParIDType_var), NumberOfParIDs := 1, Mode := mcACPAX_PARID_SET);
	IF(MC_BR_ProcessParID_AcpAx_0.Error OR MC_BR_ProcessParID_AcpAx_0.Done) THEN
		MC_BR_ProcessParID_AcpAx_Exe 			:= FALSE;
	END_IF

IF((OPCUA_R1_Down <> 0) OR (mV_R1_Down <> 0)) THEN
		OPCUA_R1_Down := 0;
		mV_R1_Down := 0;
		MC_MoveVelocity_0(Axis := ADR(gAxis_1), Execute := 1, Velocity := 30.0, Acceleration := 10.0, Deceleration := 10.0, Jerk := 0, Direction := mcPOSITIVE_DIR, BufferMode := mcABORTING);
END_IF

IF((OPCUA_R1_Up <> 0) OR (mV_R1_Up <> 0)) THEN
		OPCUA_R1_Up := 0;
		mV_R1_Up := 0;
		MC_MoveVelocity_1(Axis := ADR(gAxis_1), Execute := 1, Velocity := 30.0, Acceleration := 10.0, Deceleration := 10.0, Jerk := 0, Direction := mcNEGATIVE_DIR, BufferMode := mcABORTING);
END_IF

	IF((OPCUA_R1_Stop <> 0) OR (mV_R1_Stop <> 0)) THEN
		MC_MoveVelocity_0.Execute := FALSE;
		MC_MoveVelocity_1.Execute := FALSE;
	END_IF

	IF (MC_MoveVelocity_0.InVelocity) THEN
		OPCUA_R1_Down_Cnt := OPCUA_R1_Down_Cnt + 1;
		IF (OPCUA_R1_Down_Cnt >= 60000) THEN
			MC_MoveVelocity_0.Execute := FALSE;
		END_IF
	ELSE
		OPCUA_R1_Down_Cnt := 0;
	END_IF
	IF (MC_MoveVelocity_1.InVelocity) THEN
		OPCUA_R1_Down_Cnt := OPCUA_R1_Down_Cnt - 1;
		IF (OPCUA_R1_Down_Cnt <= 0) THEN
			MC_MoveVelocity_0.Execute := FALSE;
		END_IF
	ELSE
		OPCUA_R1_Down_Cnt := 0;
	END_IF

END_PROGRAM
```

### Program Logical/motionprg2 (IEC)

#### Variables.var
```iecst
VAR
	MpAxisBasic_0 : MpAxisBasic;
	AxisParameters : MpAxisBasicParType;
	McAcpAxProcessParIDType_var : {REDUND_UNREPLICABLE} McAcpAxProcessParIDType;
	ParId719Value : UDINT;
	MC_BR_ProcessParID_AcpAx_0 : MC_BR_ProcessParID_AcpAx;
	MC_BR_ProcessParID_AcpAx_Exe : BOOL;
	MC_MoveVelocity_0 : MC_MoveVelocity;
	MC_MoveVelocity_1 : MC_MoveVelocity;
END_VAR
```

#### Main.st
```iecst
PROGRAM _INIT

	MpAxisBasic_0.Enable := TRUE;
	MC_BR_ProcessParID_AcpAx_Exe := TRUE;

	AxisParameters.Position := 100.0;
	AxisParameters.Velocity := 10.0;
	AxisParameters.Acceleration := 50.0;
	AxisParameters.Deceleration := 50.0;
	ParId719Value := 1;
	McAcpAxProcessParIDType_var.DataType 		:= mcACPAX_PARTYPE_UDINT;
	McAcpAxProcessParIDType_var.ParID 			:= mcACPPAR_ENCOD_CMD;
	McAcpAxProcessParIDType_var.VariableAddress := ADR(ParId719Value);

END_PROGRAM

PROGRAM _CYCLIC

	MpAxisBasic_0.MpLink     := ADR(gAxis_2);
	MpAxisBasic_0.Parameters := ADR(AxisParameters);
	MpAxisBasic_0();

	MC_BR_ProcessParID_AcpAx_0(Axis := ADR(gAxis_2), Execute := MC_BR_ProcessParID_AcpAx_Exe, DataAddress := ADR(McAcpAxProcessParIDType_var), NumberOfParIDs := 1, Mode := mcACPAX_PARID_SET);
	IF(MC_BR_ProcessParID_AcpAx_0.Error OR MC_BR_ProcessParID_AcpAx_0.Done) THEN
		MC_BR_ProcessParID_AcpAx_Exe 			:= FALSE;
	END_IF

IF((OPCUA_R2_Down <> 0) OR (mV_R2_Down <> 0)) THEN
		OPCUA_R2_Down := 0;
		mV_R2_Down := 0;
		MC_MoveVelocity_0(Axis := ADR(gAxis_2), Execute := 1, Velocity := 30.0, Acceleration := 10.0, Deceleration := 10.0, Jerk := 0, Direction := mcPOSITIVE_DIR, BufferMode := mcABORTING);
END_IF

IF((OPCUA_R2_Up <> 0) OR (mV_R2_Up <> 0)) THEN
		OPCUA_R2_Up := 0;
		mV_R2_Up := 0;
		MC_MoveVelocity_1(Axis := ADR(gAxis_2), Execute := 1, Velocity := 30.0, Acceleration := 10.0, Deceleration := 10.0, Jerk := 0, Direction := mcNEGATIVE_DIR, BufferMode := mcABORTING);
END_IF

END_PROGRAM
```

### Program Logical/opctest (IEC)

#### Variables.var
```iecst
VAR
	mySinValue : REAL := 0.0;
	mySinValueIn : REAL := 0;
END_VAR
```

#### Main.st
```iecst
PROGRAM _INIT
	(* Insert code here *)
	gSchweibsChange := gSchweibsWrite;

	myDO01 := myDO02 := myDO03 := myDO04 := myDO05 := myDO06 := myDO07 := myDO08 := myDO09 := myDO10 := myDO11 := myDO12 := 0;

	mySinValue := mySinValueIn := 0;

END_PROGRAM

PROGRAM _CYCLIC
	(* Insert code here *)
	gSchweibsChange := gSchweibsChange + 1;

	mySinValueIn := mySinValueIn + 0.001;
	mySinValue := SIN(mySinValueIn);

END_PROGRAM

PROGRAM _EXIT
	(* Insert code here *)

END_PROGRAM
```

### Program Logical/room (IEC)

#### Variables.var
```iecst
VAR
	Manipulator : STRING[32];
	SwitchValue : BOOL;
	SwitchValueHW : BOOL;
	SwitchValueT : BOOL;
	SwitchValueGL : BOOL;
	SwitchValueW : BOOL;
	r_trig_0 : r_trig;
	SwitchValueTrig : BOOL;
	Lampe : BOOL;
	r_trig_HW : r_trig;
	r_trig_T : r_trig;
	r_trig_GL : r_trig;
	r_trig_W : r_trig;
	myTaskName : STRING[32];
	SendValue : BOOL;
END_VAR
VAR RETAIN
	RoomName : STRING[32];
	LampeRuntimeus : UDINT;
END_VAR
VAR
	RTInfo_0 : RTInfo;
	LampeNew : BOOL;
END_VAR
VAR RETAIN
	LampeRT : UDINT;
	LampeSwitchCnt : UDINT;
END_VAR
VAR
	tmpString : STRING[16];
END_VAR
```

#### Main.st
```iecst
PROGRAM _INIT
	(* Insert code here *)
	ST_name(0,ADR(myTaskName),0);
	RTInfo_0(enable := TRUE);
	IF(RoomName = '') THEN
		IF (myTaskName = 'room1') THEN
			RoomName := 'Kitchen';
		END_IF
		IF (myTaskName = 'room2') THEN
			RoomName := 'Living';
		END_IF
		IF (myTaskName = 'room3') THEN
			RoomName := 'Bedroom';
		END_IF
	END_IF

END_PROGRAM

PROGRAM _CYCLIC
	(* Insert code here *)

	(*raising edge*)
	r_trig_HW(CLK := SwitchValueHW);
	r_trig_T(CLK := SwitchValueT);
	r_trig_GL(CLK := SwitchValueGL);
	r_trig_W(CLK := SwitchValueW);

	(*all inputs*)
	SwitchValueTrig := r_trig_HW.Q OR r_trig_T.Q OR r_trig_GL.Q OR r_trig_W.Q;

	IF(r_trig_HW.Q) THEN
		Manipulator := 'Hardware';
	END_IF
	IF(r_trig_T.Q) THEN
		Manipulator := 'Tablett';
	END_IF
	IF(r_trig_GL.Q) THEN
		Manipulator := 'Glasses';
	END_IF
	IF(r_trig_W.Q) THEN
		Manipulator := 'Windows';
	END_IF

	(*control lamp*)
	IF (SwitchValueTrig = TRUE) THEN
		Lampe := NOT(Lampe);
		LampeSwitchCnt := LampeSwitchCnt + 1;
		gSendMessage := myTaskName;
		brsstrcat(ADR(gSendMessage), ADR('/Lampe='));
		IF (Lampe) THEN
			brsstrcat(ADR(gSendMessage), ADR('TRUE$n'));
		ELSE
			brsstrcat(ADR(gSendMessage), ADR('FALSE$n'));
		END_IF
		gDataSend := TRUE;
	END_IF
	(*tcp communication*)
	IF (SendValue = TRUE) THEN
		brsstrcat(ADR(gSendMessage), ADR(myTaskName));
		brsstrcat(ADR(gSendMessage), ADR('/Lampe='));
		IF (Lampe) THEN
			brsstrcat(ADR(gSendMessage), ADR('TRUE$n'));
		ELSE
			brsstrcat(ADR(gSendMessage), ADR('FALSE$n'));
		END_IF
		brsstrcat(ADR(gSendMessage), ADR(myTaskName));
		brsstrcat(ADR(gSendMessage), ADR('/LampeRT='));
		tmpString := UDINT_TO_STRING(LampeRT);
		brsstrcat(ADR(gSendMessage), ADR(tmpString));
		brsstrcat(ADR(gSendMessage), ADR('$n'));
		brsstrcat(ADR(gSendMessage), ADR(myTaskName));
		brsstrcat(ADR(gSendMessage), ADR('/LampeSwCnt='));
		tmpString := UDINT_TO_STRING(LampeSwitchCnt);
		brsstrcat(ADR(gSendMessage), ADR(tmpString));
		brsstrcat(ADR(gSendMessage), ADR('$n'));

		gDataSend := TRUE;
		SendValue := FALSE;
	END_IF
	IF(Lampe) THEN
		LampeRuntimeus := LampeRuntimeus + RTInfo_0.cycle_time;
		IF(LampeRuntimeus >= 1000000) THEN
			LampeRT := LampeRT + 1; // Sekunden
			LampeRuntimeus := LampeRuntimeus - 1000000;
		END_IF
	END_IF
	IF (LampeNew) THEN
		LampeNew := FALSE;
		LampeRuntimeus := 0;
		LampeRT := 0;
	END_IF

END_PROGRAM

PROGRAM _EXIT
	(* Insert code here *)

END_PROGRAM
```

### Program Logical/tcp (IEC) - Programm

#### tcp.typ
```iecst
TYPE
	room_adr : 	STRUCT
		name : STRING[80] := '::room1:SwitchValueGL';
		adr : UDINT;
		len : UDINT;
	END_STRUCT;
	CLIENT_typ : {REDUND_UNREPLICABLE} 	STRUCT
		connected : {REDUND_UNREPLICABLE} BOOL;
		data_received : {REDUND_UNREPLICABLE} BOOL;
		addr : {REDUND_UNREPLICABLE} STRING[19];
		portclnt : {REDUND_UNREPLICABLE} UINT;
		receive_buffer : {REDUND_UNREPLICABLE} ARRAY[0..255]OF USINT;
		recv : {REDUND_UNREPLICABLE} TcpRecv;
		send : {REDUND_UNREPLICABLE} TcpSend;
		close : {REDUND_UNREPLICABLE} TcpClose;
		ComTypeS : {REDUND_UNREPLICABLE} STRING[19];
		ComType : {REDUND_UNREPLICABLE} USINT;
	END_STRUCT;
END_TYPE
```

#### tcp.var
```iecst
VAR
	i : {REDUND_UNREPLICABLE} DINT;
END_VAR
VAR CONSTANT
	xERR_FUB_BUSY : UINT := 65535;
	xERR_FUB_ENABLE_FALSE : UINT := 65534;
	PORT : UINT := 8000;
	MAX_CLIENTS : USINT := 10;
	MAX_CLIENT_INDEX : USINT := MAX_CLIENTS-1;
	SERVER_OPEN : UINT := 10;
	SERVER_RUNNING : UINT := 20;
	SERVER_ERROR : UINT := 900;
END_VAR
VAR
	close : {REDUND_UNREPLICABLE} TcpClose;
	open : {REDUND_UNREPLICABLE} TcpOpen;
	server : {REDUND_UNREPLICABLE} TcpServer;
	step : {REDUND_UNREPLICABLE} UINT;
	step_str : {REDUND_UNREPLICABLE} STRING[79] := '';
	client : {REDUND_UNREPLICABLE} ARRAY[0..MAX_CLIENT_INDEX] OF CLIENT_typ;
	tempstring : {REDUND_UNREPLICABLE} STRING[79] := '';
	getipaddr : {REDUND_UNREPLICABLE} CfgGetIPAddr;
	myip : {REDUND_UNREPLICABLE} STRING[15];
	errstring : {REDUND_UNREPLICABLE} STRING[127];
	error : {REDUND_UNREPLICABLE} UINT;
END_VAR
VAR CONSTANT
	welcome_message : STRING[128] := 'Welcome TO SmartHome $nPress$n$'1$' for first message$n$'2$' for second message$n$'3$' TO abort connection$n';
	first_message : STRING[128] := 'Hi 4BHITS $n';
	second_message : STRING[128] := 'Hi Franz Schweiberer $n';
END_VAR
VAR
	lSendMessage : STRING[80];
	tmpBool : {REDUND_UNREPLICABLE} BOOL;
	SwitchValuesManager : ARRAY[0..9] OF room_adr := [(name:='::room1:SwitchValueGL'),(name:='::room1:SwitchValueT'),(name:='::room2:SwitchValueGL'),(name:='::room2:SwitchValueT'),(name:='::room3:SwitchValueGL'),(name:='::room3:SwitchValueT'),(name:='::room1:SendValue'),(name:='::room2:SendValue'),(name:='::room3:SendValue'),(0)];
	iAdr : INT;
	status_adr : UINT;
	tmpSwitch : REFERENCE TO BOOL;
	gDataSendHas : BOOL;
	HeartBeatWindows : UDINT;
	HeartBeatGlasses : UDINT;
	HeartBeatTablet : UINT;
END_VAR
```

#### tcp.st - Implementierungscode
```iecst
(*
example FOR AsTCP- library
connect with 'tcpclient.py'. Multiple connections in parallel are possible.
*)

(* startup after powerfail *)
PROGRAM _INIT

	(* this could be useful when task is overloaded... *)
	brsmemset( ADR(open), 0, SIZEOF(open) );
	brsmemset( ADR(close), 0, SIZEOF(close) );
	brsmemset( ADR(server), 0, SIZEOF(server) );
	brsmemset( ADR(getipaddr), 0, SIZEOF(getipaddr) );

	brsmemset( ADR(client), 0, SIZEOF(client) );

	server.enable := 1;

	getipaddr.enable := 1;
	getipaddr.pDevice := ADR('IF2');
	getipaddr.pIPAddr := ADR(myip);
	getipaddr.Len := SIZEOF(myip);

	step := SERVER_OPEN;

	FOR iAdr := 0 TO 9 BY 1 DO
		IF( brsstrlen(ADR(SwitchValuesManager[iAdr].name))<> 0)THEN
			status_adr := PV_xgetadr(ADR(SwitchValuesManager[iAdr].name), ADR(SwitchValuesManager[iAdr].adr), ADR(SwitchValuesManager[iAdr].len));
		END_IF
	END_FOR;
	tmpSwitch ACCESS ADR(tmpBool);

END_PROGRAM

(* cyclic code *)
PROGRAM _CYCLIC

	getipaddr();
	IF getipaddr.status = 0 THEN
		getipaddr.enable := FALSE;
	END_IF

	CASE step OF
	SERVER_OPEN:
		step_str := 'TcpOpen()';
		open.enable := TRUE;
		open.pIfAddr := 0;
		open.port := PORT;
		open.options := tcpOPT_REUSEADDR ;
		open();
		IF open.status = 0 THEN
			server.ident := open.ident;
			server.backlog := 10;
			server.pIpAddr := ADR(tempstring);
			step := SERVER_RUNNING;
		ELSIF open.status <> ERR_FUB_BUSY THEN
			errstring := 'error TcpOpen()';
			error := open.status;
			step := SERVER_ERROR;
		END_IF

	SERVER_RUNNING:
		step_str := 'server is running';
		server();
		IF  server.status = 0 THEN  (* a new client has connected *)
			FOR i := 0 TO (MAX_CLIENTS-1) DO
				IF NOT(client[i].connected)THEN
					client[i].connected := TRUE;
					client[i].addr := tempstring;
					client[i].recv.ident := server.identclnt;
					client[i].portclnt := server.portclnt;
					client[i].recv.enable := TRUE;
					client[i].recv.pData := ADR(client[i].receive_buffer);
					client[i].recv.datamax := SIZEOF(client[i].receive_buffer);
					client[i].recv.flags := 0;
					client[i].send.ident := server.identclnt;
					client[i].send.pData := ADR(welcome_message);
					client[i].send.datalen := brsstrlen(ADR(welcome_message));
					client[i].send.enable := TRUE;
					client[i].close.enable := FALSE;
					client[i].close.ident := server.identclnt;
					EXIT;
				END_IF
			END_FOR
		END_IF

		(* Noodle through all clients *)
		FOR i := 0 TO (MAX_CLIENTS-1) DO
			(* receive data... *)
			client[i].recv();

			IF client[i].recv.status = tcpERR_NOT_CONNECTED OR client[i].recv.status = tcpERR_INVALID_IDENT OR client[i].recv.status = tcpERR_SYSTEM THEN
				client[i].close.enable := TRUE;
			ELSIF client[i].recv.status = 0 THEN
				IF client[i].recv.recvlen <> 0 THEN
					client[i].data_received := TRUE; (* Flag: Data has been received *)
				ELSIF client[i].recv.recvlen = 0 THEN  (* Remote station has closed write direction *)
					client[i].close.enable := TRUE;
				END_IF
            END_IF

			(* Process input data ...*)
			IF (client[i].data_received OR (gDataSend)) AND client[i].send.enable = 0 THEN  (* Data has arrived AND send buffer is free *)
				IF (client[i].data_received) THEN
					client[i].data_received := FALSE;
					CASE client[i].receive_buffer[0] OF
						49:  (* ascii '1' *)
						client[i].send.pData := ADR(first_message);
						client[i].send.datalen := brsstrlen( client[i].send.pData );
						client[i].send.enable := TRUE;

						50: (* ascii '2' *)
						client[i].send.pData := ADR(second_message);
						client[i].send.datalen := brsstrlen( client[i].send.pData );
						client[i].send.enable := TRUE;

						51,99: (* ascii '3' *)(* ascii 'c' *)

						client[i].send.pData := ADR('bye, bye$n');
						client[i].send.datalen := brsstrlen( client[i].send.pData );
						client[i].send.enable := TRUE;
						client[i].close.enable := TRUE;

						71, 103: (*ascii 'g''G' *)
							brsmemset( ADR(lSendMessage), 0, SIZEOF(lSendMessage) );
							brsmemcpy(ADR(lSendMessage),ADR(client[i].receive_buffer),client[i].recv.recvlen);
							IF (findinstr(lSendMessage,'Glasses') = 1 OR findinstr(lSendMessage,'glasses') = 1 OR findinstr(lSendMessage,'Glass') = 1) THEN
								client[i].ComType := 1;   (*Glasses*)
								client[i].ComTypeS := 'Glasses';
								gGlassesOnline := TRUE;
							END_IF
						114,82: (* ascii 'r''R' *)
							IF(client[i].send.enable = FALSE) THEN
									brsmemset( ADR(gSendMessage), 0, SIZEOF(gSendMessage) );
									FOR iAdr := 6 TO 8 BY 1 DO
										tmpSwitch ACCESS SwitchValuesManager[iAdr].adr;
										tmpSwitch := TRUE;
									END_FOR;
									ERRxwarning(12345,i,ADR('read once message'));
								END_IF

							58,47: (* ascii : or / *)
								IF(client[i].send.enable = FALSE) THEN
									brsmemset( ADR(lSendMessage), 0, SIZEOF(lSendMessage) );
									brsmemcpy(ADR(lSendMessage),ADR(client[i].receive_buffer),client[i].recv.recvlen);
									IF (findinstr(lSendMessage,'room1') = 1 OR findinstr(lSendMessage,'room2') = 1 OR findinstr(lSendMessage,'room3') = 1) THEN
										IF (findinstr(lSendMessage,'SwitchValueGL') = 1 OR findinstr(lSendMessage,'SwitchValueT') = 1 OR findinstr(lSendMessage,'SendValue') = 1) THEN
											IF (findinstr(lSendMessage,'SwitchValueGL') = 1) THEN
												client[i].ComType := 1;   (*Glasses*)
												client[i].ComTypeS := 'Glasses';
												gGlassesOnline := TRUE;
											END_IF
											FOR iAdr := 0 TO 8 BY 1 DO
												IF( brsstrlen(ADR(SwitchValuesManager[iAdr].name))<> 0)THEN
													IF (findinstr(lSendMessage,SwitchValuesManager[iAdr].name) = 1) THEN
														tmpSwitch ACCESS SwitchValuesManager[iAdr].adr;
													END_IF
												END_IF
											END_FOR;

										IF (findinstr(lSendMessage,'True') = 1 OR findinstr(lSendMessage,'true') = 1) THEN
											brsstrcat(ADR(lSendMessage), ADR('True $n'));
											tmpSwitch := TRUE;
											gSendMessage := '';	//löschen des Sendpuffers damit leerer Puffer, wenn SendValue = True
										END_IF
										IF (findinstr(lSendMessage,'False') = 1 OR findinstr(lSendMessage,'false') = 1) THEN
											brsstrcat(ADR(lSendMessage), ADR('False $n'));
											tmpSwitch := FALSE;
										END_IF
									ELSE
											brsstrcat(ADR(lSendMessage), ADR('Back $n'));
									END_IF
								ELSE
										brsstrcat(ADR(lSendMessage), ADR('nix $n'));
								END_IF
								client[i].send.pData := ADR(lSendMessage);
								client[i].send.datalen := brsstrlen( client[i].send.pData );
								client[i].send.enable := TRUE;
								ERRxwarning(12345,i,ADR('recv message'));
							END_IF
						END_CASE
					ELSE
						IF (gDataSend) THEN
							IF((i >= MAX_CLIENTS -1) AND (gDataSendHas)) THEN
								gDataSend := FALSE;
								gDataSendHas := FALSE;
						END_IF
							IF(client[i].connected) THEN
								client[i].send.pData := ADR(gSendMessage);
								client[i].send.datalen := brsstrlen( client[i].send.pData );
								client[i].send.enable := client[i].connected;
								gDataSendHas := TRUE;
								ERRxwarning(23456,i,ADR('send message'));
							END_IF
						END_IF
				END_IF
			END_IF

			(* send output data *)
			client[i].send();
			IF client[i].send.status = 0 THEN (* sent successfully *)
				client[i].send.enable := FALSE;
			ELSIF client[i].send.status <> ERR_FUB_BUSY AND client[i].send.status <> ERR_FUB_ENABLE_FALSE THEN (* error *)
				client[i].send.enable := FALSE;
			END_IF

			(* Release socket when connection is lost *)
			client[i].close();
			IF client[i].close.enable AND client[i].close.status = 0 THEN
				IF(client[i].ComType = 1) THEN (*Glasses*)
					gGlassesOnline := FALSE;
				END_IF
				brsmemset( ADR(client[i]), 0, SIZEOF(CLIENT_typ) );
			END_IF
		END_FOR

	SERVER_ERROR:
		step_str := 'error';

	END_CASE

END_PROGRAM

(* is called on overload of the task *)
PROGRAM _EXIT

	FOR i := 0 TO (MAX_CLIENTS-1) DO
		REPEAT
			client[i].close();
			UNTIL client[i].close.status <> ERR_FUB_BUSY
		END_REPEAT
	END_FOR

	REPEAT
		close.enable := TRUE;
		close.ident := open.ident;
		close.how := 0;
		close();
		UNTIL close.status <> ERR_FUB_BUSY
	END_REPEAT

END_PROGRAM
```

Listed in the project but not available here: Logical/Global.typ, Logical/Libraries/helper/Types.typ, Logical/Libraries/helper/Constants.var
